# B&R Automation Studio project Pachore_Mayuresh_Project_3
Automation Studio 4.12.6.106; technology packages: Acp10Arnc0 5.24.1, mapp 5.24.1, mappView 5.24.4

## Configuration Config1

CPU 4PP065.0351-P74, AutomationRuntime B4.91, Build 4.1.2, Safety 1.10, Vc V4.73.2

### Task classes (Cpu.sw)
```
Cyclic#1:
  Main_Contr <- Main_Control.prg
Cyclic#2:
  Input_Brid <- Input_Bridge.prg
  Output_Bri <- Output_Bridge.prg
  Pallet <- Pallet.prg
  Crane <- Crane.prg
  Feeder <- Feeder.prg
  ComTCP_P <- Libraries.ComTCP.ComTCP_P.prg
Cyclic#4:
  Signal_Man <- Signal_Mangement.prg
Binaries: udbdef, mvLoader, FWRules, TCData, TCLang, sysconf, Role, User, iomap, ashwd, asfw, arconfig, ashwac, TC
Libraries: operator, astime, standard, AsArLog, AsBrStr, AsTCP, ComTCP_L, Signal_Mng, Gen_Axis, Gen_Device, fileio, asieccon, arssl, sys_lib, runtime, Blink, S_filter
```

### Hardware
```
4PP065_0351_P74 : 4PP065.0351-P74 v1.1.0.0
  Connector IF4:
    DNAConfiguration = manual
  Connector IF5:
    ActivateDevice = 1
  ConfigurationID = Pachore_Mayuresh_Project_3_Config1
  UserPartitionSize = 0
  Simulation = 1
  FileDevice1
  FileDeviceName1 = USER
  FileDevicePath1 = USER_PATH
  ActivateOpcUa = 1
  OpcUaInformationModels_PV_Version = 1
  KeyMappingFile = VC\4PP065_0351_P74.dis
```

### Acp10cfg.ncc - 4PP065_0351_P74/Motion/Acp10cfg.ncc
```
NcConfiguration (Version=5.24.1, NcSwId=Acp10)
  ACP10CF1_typ:
    cnt_nettrc_rec_drive = 150
    bufsize_trace_upload = 1200
    tc_nc_man_task = Cyclic #1
    glob_pv_as_ncobject = Yes
    ncsys_dl_broadcast = Yes
    ncsys_dl_acp_reset = Yes
    safemc_log_err_to_ax = Yes
    network_init:
      ncsw_init_execute = Yes
      automatic_execute = No
      node_nr_warning = Yes
      net_err_before_ncact = Yes
    nettrc:
      enter_parsecrec = Yes
      enter_ncaction = Yes
      save_ring_startidx = No
    cam_prof_download:
      cam_dat_dl_parallel = No
      tc_cam_dl_parallel = Task class for NC Manager task
```

### Acp10map.ncm - 4PP065_0351_P74/Motion/Acp10map.ncm
```
NcMapping (NcSwId=Acp10)
```

## Logical view

Binary libraries used (declarations not repeated): operator, runtime, astime, AsIecCon, Acp10man, Acp10par, NcGlobal, AsTCP, standard, AsArLog, AsBrStr, sys_lib

### MNG_Package.typ
```iecst
(*                                                                            *)
(* File generated by the B&R AS 4 control config generator                    *)
(*                                                                            *)
(*     Provider: machineering                                                 *)
(*  Application: industrialPhysics_2.4.master                                 *)
(* Architecture: Windows 64 Bit                                               *)
(*      Version: 2.4.10491.master                                             *)
(*        Build: 164f85bec                                                    *)
(*         Date: 2020-05-19, Time: 12:11:21                                   *)
(*                                                                            *)

TYPE
ComTCP_INPUTS_32BIT : STRUCT

		NumSignals	: INT := 15;

        laser_sensor_IR : BOOL := 0;
        (* BOOL laser_sensor_IR *)
        laser_sensor2_IR : BOOL := 0;
        (* BOOL laser_sensor2_IR *)
        carriage_2_AXIS : REAL := 0.0;
        (* REAL carriage_2_AXIS *)
        carriage_2_RCHD : BOOL := 0;
        (* BOOL carriage_2_RCHD *)
        turnpusher_LBK : BOOL := 0;
        (* BOOL turnpusher_LBK *)
        turnpusher_LFR : BOOL := 0;
        (* BOOL turnpusher_LFR *)
        gantry_crane_AXIS : REAL := 0.0;
        (* REAL gantry_crane_AXIS *)
        box_crane_AXIS : REAL := 0.0;
        (* REAL box_crane_AXIS *)
        vaccum_box_crane_VACUUM : BOOL := 0;
        (* BOOL vaccum_box_crane_VACUUM *)
        pallet_light_barrier_1_IR : BOOL := 0;
        (* BOOL pallet_light_barrier_1_IR *)
        pallet_light_barrier_2_IR : BOOL := 0;
        (* BOOL pallet_light_barrier_2_IR *)
        pusher_LBK : BOOL := 0;
        (* BOOL pusher_LBK *)
        pusher_LFR : BOOL := 0;
        (* BOOL pusher_LFR *)
        pallet_lifter_AXIS : REAL := 0.0;
        (* REAL pallet_lifter_AXIS *)
        pallet_fork_left_FB : BOOL := 0;
        (* BOOL pallet_fork_left_FB *)

	END_STRUCT;

ComTCP_OUTPUTS_32BIT : STRUCT

		NumSignals	: INT := 18;

        cartboard_TRIG : BOOL := 0;
        (* BOOL cartboard_TRIG *)
        conveyor_if_FWD : BOOL := 0;
        (* BOOL conveyor_if_FWD *)
        conveyer_turn1_FWD : BOOL := 0;
        (* BOOL conveyer_turn1_FWD *)
        conveyer_end_FWD : BOOL := 0;
        (* BOOL conveyer_end_FWD *)
        carriage_2_TGT_POS : REAL := 0.0;
        (* REAL carriage_2_TGT_POS *)
        turnpusher_FWD : BOOL := 0;
        (* BOOL turnpusher_FWD *)
        turnpusher_BWD : BOOL := 0;
        (* BOOL turnpusher_BWD *)
        gantry_crane_TGT_POS : REAL := 0.0;
        (* REAL gantry_crane_TGT_POS *)
        box_crane_TGT_POS : REAL := 0.0;
        (* REAL box_crane_TGT_POS *)
        slide_rail_right_EN : BOOL := 0;
        (* BOOL slide_rail_right_EN *)
        vaccum_box_crane_GRIP : BOOL := 0;
        (* BOOL vaccum_box_crane_GRIP *)
        pusher_z_EN : BOOL := 0;
        (* BOOL pusher_z_EN *)
        pusher_x_EN : BOOL := 0;
        (* BOOL pusher_x_EN *)
        pallet_conveyor_2_ACT_VEL : REAL := 0.0;
        (* REAL pallet_conveyor_2_ACT_VEL *)
        pusher_FW : BOOL := 0;
        (* BOOL pusher_FW *)
        pallet_lifter_TGT_POS : REAL := 0.0;
        (* REAL pallet_lifter_TGT_POS *)
        pallet_fork_left_EN : BOOL := 0;
        (* BOOL pallet_fork_left_EN *)
        pallet_conveyor_1_FWD : BOOL := 0;
        (* BOOL pallet_conveyor_1_FWD *)

	END_STRUCT;

END_TYPE
```

### MNG_Package.var
```iecst
(*                                                                            *)
(* File generated by the B&R AS 4 control config generator                    *)
(*                                                                            *)
(*     Provider: machineering                                                 *)
(*  Application: industrialPhysics_2.4.master                                 *)
(* Architecture: Windows 64 Bit                                               *)
(*      Version: 2.4.10491.master                                             *)
(*        Build: 164f85bec                                                    *)
(*         Date: 2020-05-19, Time: 12:11:21                                   *)
(*                                                                            *)

                VAR
                ComTCP_SimInputs : ComTCP_INPUTS_32BIT := (0);
    ComTCP_SimOutputs : ComTCP_OUTPUTS_32BIT := (0);

    ComTCP_SimServerAddress : STRING[15] := '127.0.0.1';
    ComTCP_SimServerPort : UINT := 5000;
    ComTCP_SimSendCycleTime : TIME := T#5ms;
    ComTCP_SimActive : BOOL := FALSE;

                END_VAR
```

### Global.var - Global variables
```iecst
(*Simulation Variables*)
(*Input Variables*)
VAR
	I_IR_Sensor_1 : BOOL := FALSE; (*laser_sensor_IR*)
	I_IR_Sensor_2 : BOOL := FALSE; (*laser_sensor2_IR*)
	I_Carriage_Push_Act_Pos : REAL := 1; (*carriage_2_AXIS*)
	I_Carriage_Push_Tar_Rec : BOOL := TRUE; (*carriage_2_RCHD*)
	I_Pusher_1_B : BOOL := FALSE; (*pusher_LBK*)
	I_Pusher_1_F : BOOL := TRUE; (*pusher_LFR*)
	I_Turn_Push_B : BOOL := FALSE; (*turnpusher_LBK*)
	I_Turn_Push_F : BOOL := TRUE; (*turnpusher_LFR*)
	I_Gantry_Crane_Act_Pos : REAL := 0; (*gantry_crane_AXIS*)
	I_Box_Crane_Act_Pos : REAL := 0; (*box_crane_AXIS*)
	I_Vacuum_retention_act : BOOL := FALSE; (*vacuum_box_crane_VACUUM*)
	I_Pallet_lift_Act_Pos : REAL := 0; (*pallet_lifter_AXIS*)
	I_Pallet_holder_State : BOOL := FALSE; (*pallet_fork_left_FB*)
	I_IR_Sensor_3 : BOOL := FALSE; (*pallet_light_barrier_1_IR*)
	I_IR_Sensor_4 : BOOL := FALSE; (*pallet_light_barrier_2_IR*)
END_VAR
(*Output Variables*)
VAR
	O_Conveyor_1 : BOOL := FALSE; (*Conveyor_if control*)
	O_Pusher_1 : BOOL := FALSE; (*pusher control*)
	O_Conveyor_2 : BOOL := FALSE; (*conveyor_turn1 control*)
	O_Conveyor_3 : BOOL := FALSE; (*conveyor_end control*)
	O_Turn_Pusher_ON : BOOL := FALSE; (*turnpusher Forward*)
	O_Turn_Pusher_OFF : BOOL := FALSE; (*turnpusher Backward*)
	O_Carriage_Tar_Pos : REAL := 0; (*carriage_2 control*)
	O_Gantry_Crane_Tar_Pos : REAL := 0; (*gantry_crane control*)
	O_Box_Crane_Tar_Pos : REAL := 0; (*box_crane control*)
	O_Cartboard_Trig : BOOL := FALSE; (*cartboard control*)
	O_Vacuum_Grip_act : BOOL := FALSE; (*vacuum_box_crane control*)
	O_Box_Holder : BOOL := FALSE; (*slide_rail_right control*)
	O_Pusher_z : BOOL := FALSE; (*pusher_z control*)
	O_Pusher_x : BOOL := FALSE; (*pusher_x control*)
	O_Pallet_lift_Tar_Pos : REAL := 0; (*pallet_lifter control*)
	O_Pallet_Holder : BOOL := FALSE; (*pallet_fork control*)
	O_Conveyor_4 : BOOL := FALSE; (*pallet_conveyor_1 control*)
	O_Conveyor_5_vel : REAL := 0; (*pallet_conveyor_2 control*)
END_VAR
(*HMI Variables*)
VAR
	Service_Mode_HMI : BOOL;
	Conveyor_1_Jog_HMI : BOOL;
	Pusher_1_Jog_HMI : BOOL;
	Conveyor_2_Jog_HMI : BOOL;
	Conveyor_3_Jog_HMI : BOOL;
	Conveyor_1_HMI : BOOL;
	Pusher_1_HMI : BOOL;
	Conveyor_2_HMI : BOOL;
	Conveyor_3_HMI : BOOL;
	Turn_Pusher_ON_HMI : BOOL;
	Turn_Pusher_OFF_HMI : BOOL;
	Carriage_Push_Origin_HMI : BOOL;
	Carriage_Push_Target_HMI : BOOL;
	Carriage_Target_Pos_HMI : REAL;
	Carriage_Tar_Pos_Dis_HMI : REAL;
	IR1_HMI : BOOL;
	IR2_HMI : BOOL;
	Turn_Pusher_F_HMI : BOOL;
	Turn_Pusher_B_HMI : BOOL;
	Pusher_1_F_HMI : BOOL;
	Pusher_1_B_HMI : BOOL;
	Carriage_Push_TarRech_HMI : BOOL;
	Carriage_Push_ActPos_Dis_HMI : REAL;
	vaccume_box_crane_grip_HMI : BOOL;
	Cartboard_Trig_HMI : BOOL;
	Slide_rail_right_EN_HMI : BOOL;
	pusher_z_EN_HMI : BOOL;
	pusher_x_EN_HMI : BOOL;
	gantry_crane_Origin_pos_HMI : BOOL;
	gantry_crane_TGT_pos_HMI : BOOL;
	gantry_crane_TGT_HMI : REAL;
	gantry_crane_TGT_dis_HMI : REAL;
	box_crane_TGT_pos_HMI : BOOL;
	box_crane_Origin_pos_HMI : BOOL;
	box_crane_TGT_HMI : REAL;
	box_crane_TGT_dis_HMI : REAL;
	vaccume_box_crane_state_HMI : BOOL;
	gantry_crane_Act_Pos_HMI : REAL;
	box_crane_Act_Pos_HMI : REAL;
	Pallet_fork_HMI : BOOL;
	Conveyor_4_Jog_HMI : BOOL;
	Conveyor_4_HMI : BOOL;
	Conveyor_5_S1_HMI : BOOL;
	Conveyor_5_S2_HMI : BOOL;
	Pallet_Lifter_Origin_pos_HMI : BOOL;
	Pallet_Lifter_TGT_pos_HMI : BOOL;
	Pallet_Lifter_TGT_HMI : REAL;
	Pallet_Lifter_TGT_dis_HMI : REAL;
	Pallet_Holder_State_HMI : BOOL;
	IR_3_HMI : BOOL;
	IR_4_HMI : BOOL;
	On_Phase_Stop_HMI : BOOL;
	Emergency_Stop_HMI : BOOL;
	Priority_4_HMI : STRING[80];
	Priority_3_HMI : STRING[80];
	Priority_2_HMI : STRING[80];
	Priority_1_HMI : STRING[80];
	Pallet_Lifter_Act_Pos_HMI : REAL;
END_VAR
(*Signal_Mng_Faults*)
VAR
	Operation_Type : INT := 0;
	Out_Of_Material : BOOL;
	Crane_Cartboard_Counter : INT := 3;
	Pallet_Counter : INT := 5;
	e_Turn_Pusher_Fault : BOOL := FALSE;
	e_Feeder_Pusher_Fault : BOOL := FALSE;
	e_Crane_Pusher_x_Fault : BOOL := FALSE;
	e_Crane_Pusher_z_Fault : BOOL := FALSE;
	e_Vacuum_Fault : BOOL := FALSE;
	e_Pallet_Fork_Fault : BOOL := FALSE;
	e_Carriage_Fault : BOOL := FALSE;
	e_Gantry_Crane_Fault : BOOL := FALSE;
	e_Box_Crane_Fault : BOOL := FALSE;
	e_Pallet_Lifter_Fault : BOOL := FALSE;
	e_Conveyor_1_Fault : BOOL := FALSE;
	e_Conveyor_2_Fault : BOOL := FALSE;
	e_Conveyor_3_Fault : BOOL := FALSE;
	e_Cartboard_Fault : BOOL := FALSE;
	e_Box_Holder_Fault : BOOL := FALSE;
	e_Conveyor_4_Fault : BOOL := FALSE;
	e_Conveyor_5_Fault : BOOL := FALSE;
	Fault : ARRAY[0..23] OF STRING[80] := ['',2('Feeder Fault Technician Required'),3('Crane Fault Technician Required'),'Pallet Fault Technician Required','Pallet Refill Required','Feeder Fault Technician Required',2('Crane Fault Technician Required'),'Pallet Fault Technician Required','Prepare Pallets to Refill','On Phase Stop Requested','Emergency Stop Requested','Prepare Cartboards to Refill','Cartboard Refill Required',3('Feeder Fault Technician Required'),2('Crane Fault Technician Required'),2('Pallet Fault Technician Required')];
END_VAR
(*Main*)
VAR
	Service_Mode : BOOL;
	En_Machine : BOOL := FALSE;
	Start_Machine : BOOL := FALSE;
	Emergency_Stop : BOOL;
	Immediate_Stop : BOOL;
	On_Phase_Stop : BOOL;
	Hold_Boxes : BOOL;
	P_Exit_Done : BOOL;
	Boxes_On_The_P : BOOL;
	Boxes_On_The_C : BOOL; (*Feeder*)
	Load_Boxes_On_The_C : BOOL; (*Feeder*)
	Load_Boxes_On_The_P : BOOL;
	Second_Layer : BOOL; (*Feeder*)
	M_Current_State : STRING[80];
	P_Exit_En : BOOL;
END_VAR
(*Communication between Feeder and Main*)
VAR
	Start_Feeder : BOOL := FALSE;
	F_Emergency_Stop : BOOL := FALSE;
	F_Reset_Config : BOOL := FALSE;
	F_Immediate_Stop : BOOL := FALSE;
	F_On_Phase_Stop : BOOL := FALSE;
	F_Restart : BOOL := FALSE;
	F_Ready : BOOL := FALSE;
END_VAR
(*Communication between Crane and Main*)
VAR
	Start_Crane : BOOL := FALSE;
	C_Reset_Config : BOOL := FALSE;
	C_Emergency_Stop : BOOL := FALSE;
	C_Immediate_Stop : BOOL := FALSE;
	C_On_Phase_Stop : BOOL := FALSE;
	C_Restart : BOOL := FALSE;
	C_Ready : BOOL := FALSE;
END_VAR
(*Communication between Pallet and Main*)
VAR
	Start_Pallet : BOOL := FALSE;
	P_Emergency_Stop : BOOL := FALSE;
	P_Reset_Config : BOOL := FALSE;
	P_Immediate_Stop : BOOL := FALSE;
	P_On_Phase_Stop : BOOL := FALSE;
	P_Restart : BOOL := FALSE;
	P_Ready : BOOL := FALSE;
END_VAR
(*Feeder Variables*)
VAR
	Conveyor_3_Fault_HMI : BOOL;
	Conveyor_2_Fault_HMI : BOOL;
	Conveyor_1_Fault_HMI : BOOL;
	Turn_Pusher_Fault_HMI : BOOL;
	Carriage_Fault_HMI : BOOL;
	Pusher_1_Fault_HMI : BOOL;
	Box_Counter : INT := 0;
	C_Layer_Counter : BOOL := FALSE;
	End_Layer : BOOL;
	F_Current_State : STRING[80];
END_VAR
(*Crane Variables*)
VAR
	Gantry_Crane_Fault_HMI : BOOL;
	Box_Crane_Fault_HMI : BOOL;
	Cartboard_Fault_HMI : BOOL;
	Vacuum_Fault_HMI : BOOL;
	Box_Holder_Fault_HMI : BOOL;
	Crane_Pusher_X_Fault_HMI : BOOL;
	Crane_Pusher_Z_Fault_HMI : BOOL;
	C_Current_State : STRING[80];
END_VAR
(*Pallet Variables*)
VAR
	Pallet_Lifter_Fault_HMI : BOOL;
	Pallet_Fork_Fault_HMI : BOOL;
	Pallet_Conv_1_Fault_HMI : BOOL;
	Pallet_Conv_2_Fault_HMI : BOOL;
	P_Current_State : STRING[80];
END_VAR
(*LED Blinker*)
VAR
	Reset_Unlocked : BOOL;
	Aux_Reset_Unlocked : BOOL;
	Aux_Unlocked : Blink;
	R_Unlocked : Blink;
	Warning_Detected : Blink;
	Alarm_Detected : Blink;
END_VAR
```

### Package Logical/Libraries - Global libraries

### Library Logical/Libraries/ComTCP/ComTCP_L (ANSIC)
Depends on: AsTCP, operator, runtime, astime, standard, AsArLog, AsBrStr, Convert

#### MNG_ComHdlr.hpp
```cpp
#ifndef _MNGCOMHDLR_HPP_
#define _MNGCOMHDLR_HPP_

#define TRUE  1
#define FALSE 0

#include "MNG_InternalTyp.hpp"

#include <bur/plc.h>
#include <bur/plctypes.h>
#include <AsTCP.h>
#include <standard.h>
#include <astime.h>
#include <runtime.h>
#include <AsBrStr.h>

typedef struct{
	TcpOpen_typ tcpOpen;
	TcpIoctl_typ tcpIoctl;
	tcpLINGER_typ tcpLINGER;
	TcpSend_typ tcpSend;
	TcpClose_typ tcpClose;
	TcpRecv_typ tcpRecv;
	TcpClient_typ tcpClient;
} asTcpFcn_t;

typedef enum {
	MNG_wSock,
	MNG_skippedMessage
} MNG_errorCases;

typedef enum {
	MNG_Init,
	MNG_Socket,
	MNG_Open,
	MNG_SetIo,
	MNG_Linger,
	MNG_Connecting,
	MNG_Exchange,
	MNG_Closing,
        MNG_Reset
} MNG_internalState_t;

	extern unsigned long int MNG_CpyOutToMsg(MNG_RawDatagram * pToServer, unsigned long int counter, ComTCP_OUTPUTS_32BIT_FWRD *pSimOutputs);
	extern unsigned long int MNG_CpyMsgToInp(MNG_RawDatagram * pFromServer, ComTCP_INPUTS_32BIT_FWRD *pSimInputs);

class MNG_ComHdlr
{
	public:

	MNG_ComHdlr(char *srvIpAdr, unsigned int srvPort, TIME sendCycleTime);
	~MNG_ComHdlr();

        int RunCommunication(void*, void*, BOOL*);

	private:

	char* _srvIpAdr;
	unsigned int _srvPort;
	TIME _sendCycleTime;

	unsigned int _error;

	MNG_internalState_t _internalState;
	TON_typ _connectionTon;
	TIME _connectionTime;

	bool _connect;
	bool _sendDone;

	signed int _recvOffset;

	signed long int _potMsgLen;
	signed long int _totalRecvLen;

	unsigned long int _one;
	unsigned long int _counter;
	unsigned long int _recvLen;
	unsigned long int _recvBuffer[10000];
	TON_typ _sendTon;
	MNG_RawDatagram _recvMessage;
	MNG_RawDatagram _sendMessage;

	static const signed long int SIXTEEN = 16;
	static const unsigned int PORT = 0;
	static const unsigned long int MNG_MAXPAYLOAD = 1400;

	void init_TcpOpen();
	void init_TcpSocket();
	void init_TcpIoctl();
	void init_TcpLinger();
	void init_TcpClient();
	void init_TcpRecv();
	void init_TcpSend(ComTCP_OUTPUTS_32BIT_FWRD* pSimOut);

	void InitParams();

	void SetSendDone(bool toogle);
	void SetStateValue(MNG_internalState_t stateVal);

};
#endif
```

#### MNG_Global.hpp
```cpp
#ifndef  _MNGGLOBAL_HPP_
#define _MNGGLOBAL_HPP_

#include <mng_globalTYP.h>

    typedef struct {

		signed short NumSignals;

        /* BOOL laser_sensor_IR */
        BOOL laser_sensor_IR;
        /* BOOL laser_sensor2_IR */
        BOOL laser_sensor2_IR;
        /* REAL carriage_2_AXIS */
        REAL carriage_2_AXIS;
        /* BOOL carriage_2_RCHD */
        BOOL carriage_2_RCHD;
        /* BOOL turnpusher_LBK */
        BOOL turnpusher_LBK;
        /* BOOL turnpusher_LFR */
        BOOL turnpusher_LFR;
        /* REAL gantry_crane_AXIS */
        REAL gantry_crane_AXIS;
        /* REAL box_crane_AXIS */
        REAL box_crane_AXIS;
        /* BOOL vaccum_box_crane_VACUUM */
        BOOL vaccum_box_crane_VACUUM;
        /* BOOL pallet_light_barrier_1_IR */
        BOOL pallet_light_barrier_1_IR;
        /* BOOL pallet_light_barrier_2_IR */
        BOOL pallet_light_barrier_2_IR;
        /* BOOL pusher_LBK */
        BOOL pusher_LBK;
        /* BOOL pusher_LFR */
        BOOL pusher_LFR;
        /* REAL pallet_lifter_AXIS */
        REAL pallet_lifter_AXIS;
        /* BOOL pallet_fork_left_FB */
        BOOL pallet_fork_left_FB;

        } ComTCP_INPUTS_32BIT_FWRD;

    typedef struct {

		signed short NumSignals;

        /* BOOL cartboard_TRIG */
        BOOL cartboard_TRIG;
        /* BOOL conveyor_if_FWD */
        BOOL conveyor_if_FWD;
        /* BOOL conveyer_turn1_FWD */
        BOOL conveyer_turn1_FWD;
        /* BOOL conveyer_end_FWD */
        BOOL conveyer_end_FWD;
        /* REAL carriage_2_TGT_POS */
        REAL carriage_2_TGT_POS;
        /* BOOL turnpusher_FWD */
        BOOL turnpusher_FWD;
        /* BOOL turnpusher_BWD */
        BOOL turnpusher_BWD;
        /* REAL gantry_crane_TGT_POS */
        REAL gantry_crane_TGT_POS;
        /* REAL box_crane_TGT_POS */
        REAL box_crane_TGT_POS;
        /* BOOL slide_rail_right_EN */
        BOOL slide_rail_right_EN;
        /* BOOL vaccum_box_crane_GRIP */
        BOOL vaccum_box_crane_GRIP;
        /* BOOL pusher_z_EN */
        BOOL pusher_z_EN;
        /* BOOL pusher_x_EN */
        BOOL pusher_x_EN;
        /* REAL pallet_conveyor_2_ACT_VEL */
        REAL pallet_conveyor_2_ACT_VEL;
        /* BOOL pusher_FW */
        BOOL pusher_FW;
        /* REAL pallet_lifter_TGT_POS */
        REAL pallet_lifter_TGT_POS;
        /* BOOL pallet_fork_left_EN */
        BOOL pallet_fork_left_EN;
        /* BOOL pallet_conveyor_1_FWD */
        BOOL pallet_conveyor_1_FWD;

        } ComTCP_OUTPUTS_32BIT_FWRD;

#endif
```

#### MNG_CpyOutToMsg.cpp
```cpp
#include "MNG_InternalTyp.hpp"

unsigned long int MNG_CpyOutToMsg(MNG_RawDatagram * pToServer, unsigned long int counter, ComTCP_OUTPUTS_32BIT_FWRD *pSimOutputs ) {

        unsigned long int DWordBuffer;

        pSimOutputs->NumSignals = 18;
        (pToServer->Header).ByteCount    = H_TO_NUDINT(76);
        (pToServer->Header).DatagramType = H_TO_NUDINT(MNG_Raw32BitImage);
        (pToServer->Header).SentTime = H_TO_NUDINT(0);  // Todo
        (pToServer->Header).Counter = H_TO_NUDINT(counter);
        pToServer->Payload[0] = H_TO_NUDINT(pSimOutputs->NumSignals);

    /* cartboard_TRIG : BOOL */
    if(pSimOutputs->cartboard_TRIG == 1) {
        pToServer->Payload[1] = 0xFFFFFFFF;   /*BOOL */
    } else {
        pToServer->Payload[1] = 0;
    }

    /* conveyor_if_FWD : BOOL */
    if(pSimOutputs->conveyor_if_FWD == 1) {
        pToServer->Payload[2] = 0xFFFFFFFF;   /*BOOL */
    } else {
        pToServer->Payload[2] = 0;
    }

    /* conveyer_turn1_FWD : BOOL */
    if(pSimOutputs->conveyer_turn1_FWD == 1) {
        pToServer->Payload[3] = 0xFFFFFFFF;   /*BOOL */
    } else {
        pToServer->Payload[3] = 0;
    }

    /* conveyer_end_FWD : BOOL */
    if(pSimOutputs->conveyer_end_FWD == 1) {
        pToServer->Payload[4] = 0xFFFFFFFF;   /*BOOL */
    } else {
        pToServer->Payload[4] = 0;
    }

    /* carriage_2_TGT_POS : FLOAT32 */
    brsmemcpy((unsigned long int)&(DWordBuffer), (unsigned long int)&(pSimOutputs->carriage_2_TGT_POS), 4);
    pToServer->Payload[5] = H_TO_NUDINT(DWordBuffer);

    /* turnpusher_FWD : BOOL */
    if(pSimOutputs->turnpusher_FWD == 1) {
        pToServer->Payload[6] = 0xFFFFFFFF;   /*BOOL */
    } else {
        pToServer->Payload[6] = 0;
    }

    /* turnpusher_BWD : BOOL */
    if(pSimOutputs->turnpusher_BWD == 1) {
        pToServer->Payload[7] = 0xFFFFFFFF;   /*BOOL */
    } else {
        pToServer->Payload[7] = 0;
    }

    /* gantry_crane_TGT_POS : FLOAT32 */
    brsmemcpy((unsigned long int)&(DWordBuffer), (unsigned long int)&(pSimOutputs->gantry_crane_TGT_POS), 4);
    pToServer->Payload[8] = H_TO_NUDINT(DWordBuffer);

    /* box_crane_TGT_POS : FLOAT32 */
    brsmemcpy((unsigned long int)&(DWordBuffer), (unsigned long int)&(pSimOutputs->box_crane_TGT_POS), 4);
    pToServer->Payload[9] = H_TO_NUDINT(DWordBuffer);

    /* slide_rail_right_EN : BOOL */
    if(pSimOutputs->slide_rail_right_EN == 1) {
        pToServer->Payload[10] = 0xFFFFFFFF;   /*BOOL */
    } else {
        pToServer->Payload[10] = 0;
    }

    /* vaccum_box_crane_GRIP : BOOL */
    if(pSimOutputs->vaccum_box_crane_GRIP == 1) {
        pToServer->Payload[11] = 0xFFFFFFFF;   /*BOOL */
    } else {
        pToServer->Payload[11] = 0;
    }

    /* pusher_z_EN : BOOL */
    if(pSimOutputs->pusher_z_EN == 1) {
        pToServer->Payload[12] = 0xFFFFFFFF;   /*BOOL */
    } else {
        pToServer->Payload[12] = 0;
    }

    /* pusher_x_EN : BOOL */
    if(pSimOutputs->pusher_x_EN == 1) {
        pToServer->Payload[13] = 0xFFFFFFFF;   /*BOOL */
    } else {
        pToServer->Payload[13] = 0;
    }

    /* pallet_conveyor_2_ACT_VEL : FLOAT32 */
    brsmemcpy((unsigned long int)&(DWordBuffer), (unsigned long int)&(pSimOutputs->pallet_conveyor_2_ACT_VEL), 4);
    pToServer->Payload[14] = H_TO_NUDINT(DWordBuffer);

    /* pusher_FW : BOOL */
    if(pSimOutputs->pusher_FW == 1) {
        pToServer->Payload[15] = 0xFFFFFFFF;   /*BOOL */
    } else {
        pToServer->Payload[15] = 0;
    }

    /* pallet_lifter_TGT_POS : FLOAT32 */
    brsmemcpy((unsigned long int)&(DWordBuffer), (unsigned long int)&(pSimOutputs->pallet_lifter_TGT_POS), 4);
    pToServer->Payload[16] = H_TO_NUDINT(DWordBuffer);

    /* pallet_fork_left_EN : BOOL */
    if(pSimOutputs->pallet_fork_left_EN == 1) {
        pToServer->Payload[17] = 0xFFFFFFFF;   /*BOOL */
    } else {
        pToServer->Payload[17] = 0;
    }

    /* pallet_conveyor_1_FWD : BOOL */
    if(pSimOutputs->pallet_conveyor_1_FWD == 1) {
        pToServer->Payload[18] = 0xFFFFFFFF;   /*BOOL */
    } else {
        pToServer->Payload[18] = 0;
    }

	return 0;
}
```

#### MNG_CpyMsgToInp.cpp
```cpp
#include "MNG_InternalTyp.hpp"

unsigned long int MNG_CpyMsgToInp(MNG_RawDatagram * pFromServer, ComTCP_INPUTS_32BIT_FWRD *pSimInputs) {

    MNG_DatagramType datagramType;
	unsigned long int DWordBuffer;
        unsigned long int byteCount;
	unsigned long int numSignalsInMessage;

	byteCount = N_TO_HUDINT((pFromServer->Header).ByteCount);
	datagramType = static_cast<MNG_DatagramType>(N_TO_HUDINT((pFromServer->Header).DatagramType));
	if (datagramType != MNG_Raw32BitImage) {
		return 0;
	}

    pSimInputs->NumSignals = 15;

    numSignalsInMessage = N_TO_HUDINT(pFromServer->Payload[0]);
        if ((static_cast<long int>(numSignalsInMessage) != pSimInputs->NumSignals) ||
	(byteCount != 4 + numSignalsInMessage * 4)) {
		return 0;
	}

    /* BOOL laser_sensor_IR */
    pSimInputs->laser_sensor_IR = (pFromServer->Payload[1] != 0);

    /* BOOL laser_sensor2_IR */
    pSimInputs->laser_sensor2_IR = (pFromServer->Payload[2] != 0);

    /* FLOAT32 carriage_2_AXIS */
    DWordBuffer = N_TO_HUDINT(pFromServer->Payload[3]);
    brsmemcpy((unsigned long int)&(pSimInputs->carriage_2_AXIS), (unsigned long int)&(DWordBuffer), 4);

    /* BOOL carriage_2_RCHD */
    pSimInputs->carriage_2_RCHD = (pFromServer->Payload[4] != 0);

    /* BOOL turnpusher_LBK */
    pSimInputs->turnpusher_LBK = (pFromServer->Payload[5] != 0);

    /* BOOL turnpusher_LFR */
    pSimInputs->turnpusher_LFR = (pFromServer->Payload[6] != 0);

    /* FLOAT32 gantry_crane_AXIS */
    DWordBuffer = N_TO_HUDINT(pFromServer->Payload[7]);
    brsmemcpy((unsigned long int)&(pSimInputs->gantry_crane_AXIS), (unsigned long int)&(DWordBuffer), 4);

    /* FLOAT32 box_crane_AXIS */
    DWordBuffer = N_TO_HUDINT(pFromServer->Payload[8]);
    brsmemcpy((unsigned long int)&(pSimInputs->box_crane_AXIS), (unsigned long int)&(DWordBuffer), 4);

    /* BOOL vaccum_box_crane_VACUUM */
    pSimInputs->vaccum_box_crane_VACUUM = (pFromServer->Payload[9] != 0);

    /* BOOL pallet_light_barrier_1_IR */
    pSimInputs->pallet_light_barrier_1_IR = (pFromServer->Payload[10] != 0);

    /* BOOL pallet_light_barrier_2_IR */
    pSimInputs->pallet_light_barrier_2_IR = (pFromServer->Payload[11] != 0);

    /* BOOL pusher_LBK */
    pSimInputs->pusher_LBK = (pFromServer->Payload[12] != 0);

    /* BOOL pusher_LFR */
    pSimInputs->pusher_LFR = (pFromServer->Payload[13] != 0);

    /* FLOAT32 pallet_lifter_AXIS */
    DWordBuffer = N_TO_HUDINT(pFromServer->Payload[14]);
    brsmemcpy((unsigned long int)&(pSimInputs->pallet_lifter_AXIS), (unsigned long int)&(DWordBuffer), 4);

    /* BOOL pallet_fork_left_FB */
    pSimInputs->pallet_fork_left_FB = (pFromServer->Payload[15] != 0);

return N_TO_HUDINT((pFromServer->Header).Counter); // return counter
}
```

### Program Logical/Libraries/ComTCP/ComTCP_P

#### Main.cpp
```cpp
#include <bur/plctypes.h>

#ifdef _DEFAULT_INCLUDES
        #include <AsDefault.h>
#endif

#include "../ComTCP_L/MNG_Global.hpp"
#include "../ComTCP_L/MNG_InternalTyp.hpp"
#include "../ComTCP_L/MNG_ComHdlr.hpp"

unsigned long bur_heap_size = 0xFFFF;

MNG_ComHdlr *pMNG_ComHdlr;

void _INIT ProgramInit(void)
{
    pMNG_ComHdlr = new MNG_ComHdlr(ComTCP_SimServerAddress, ComTCP_SimServerPort, ComTCP_SimSendCycleTime);
}

void _CYCLIC ProgramCyclic(void)
{
    connectionState = pMNG_ComHdlr->RunCommunication((void*)&ComTCP_SimInputs,(void*)&ComTCP_SimOutputs, &ComTCP_SimActive);
}

void _EXIT ProgramExit(void)
{
    delete pMNG_ComHdlr;
}
```

### Library Logical/Libraries/S_filter (IEC)

#### S_filter.fun - Exported functions and function blocks
```iecst
FUNCTION_BLOCK S_filter
	VAR_INPUT
		Sensor_Raw : BOOL;
		Sensor_Data : REAL;
		threshold_F : REAL;
		threshold_B : INT;
		Is_Bool : BOOL;
	END_VAR
	VAR_OUTPUT
		Sensor_Filtered : BOOL;
		Sensor_Data_Filtered : REAL;
	END_VAR
	VAR
		last_State : BOOL := FALSE;
		counter : INT := 0;
		init : BOOL := FALSE;
	END_VAR
END_FUNCTION_BLOCK
```

#### S_filter.st
```iecst
(* For Sensor Data Filter *)
FUNCTION_BLOCK S_filter
	IF Is_Bool THEN
		// BOOLEAN MODE filtering
		IF Sensor_Raw = last_State THEN
			counter := counter + 1;
		ELSE
			counter := 0;
			last_State := Sensor_Raw;
		END_IF;

		IF counter >= threshold_B THEN
			Sensor_Filtered := Sensor_Raw;
			counter := 0; // reset after output change
		END_IF;

	ELSE
		// REAL MODE: Exponential smoothing
		IF NOT init THEN
			Sensor_Data_Filtered := Sensor_Data;
			init := TRUE;
		ELSE
			Sensor_Data_Filtered := threshold_F * Sensor_Data + (1.0 - threshold_F) * Sensor_Data_Filtered;
		END_IF;
	END_IF;

END_FUNCTION_BLOCK
```

### Library Logical/Libraries/Signal_Mng (IEC)

#### Constants.var - Exported constants
```iecst
VAR CONSTANT
	Init : INT := 0;
	Run : INT := 1;
	Start_Configuration : INT := 2;
	Configuration : INT := 3;
	Start_Generation : INT := 4;
	Generation : INT := 5;
	Alarm : DINT := 2#0000000000000001;
	Anomaly : DINT := 2#0000000000000010;
	Warning : DINT := 2#0000000000000011;
	Information : DINT := 2#0000000000000100;
	Aux_Reset : DINT := 2#0000001000000000;
	Unconditioned_Reset : DINT := 2#0100000000000000;
	Auto_Conditioned_Reset : DINT := 2#0010000000000000;
	Auto_Provisional_Reset : DINT := 2#0001000000000000;
	Auto_Priority_Reset : DINT := 2#0000100000000000;
	Auto_Reset : DINT := 2#0000010000000000;
	Signal_Type_Mask : DINT := 2#0000000000000111;
	Sign_None : DWORD := 16#0000;
	Sign_Emergency_Stop : DWORD := 16#0001;
	Sign_Immediate_Stop : DWORD := 16#0002;
	Sign_On_Phase_Stop : DWORD := 16#0004;
	Sign_Machine_Out_Of_Phase : DWORD := 16#0100;
	Sign_Machine_Inhibition : DWORD := 16#0200;
	Sign_Materials_Run_Out_Lamp : DWORD := 16#0400;
	Sign_Materials_Run_Out_Buzzer : DWORD := 16#0800;
	Sign_IO_Diagostic_Inhibition : DWORD := 16#8000;
END_VAR
```

#### Signal_Mng.fun - Exported functions and function blocks
```iecst
FUNCTION_BLOCK Signal_Mng
	VAR_INPUT
		Operation_Type : INT;
		Signal_Type : DINT := 0;
		Signal_Code : INT := 0;
		Signal_Output : DWORD := 0;
		Activation_Signal : BOOL := FALSE;
		Auto_Reset_Signal : BOOL := FALSE;
		Reset : BOOL;
		Key_Reset : BOOL;
	END_VAR
	VAR_OUTPUT
		Signal_Outputs : DWORD;
		Signal_Priority_Code : WORD;
		Reset_Enable : BOOL;
		Aux_Reset_Enable : BOOL;
		Signal_Type_Alarm : BOOL;
		Signal_Type_Anomaly : BOOL;
		Signal_Type_Warning : BOOL;
		Signal_Type_Information : BOOL;
		Number_of_Alarms : INT;
		Number_of_Anomalies : INT;
		Number_of_Warnings : INT;
		Number_of_Information : INT;
		Active_Signal_Codes : ARRAY[1..30] OF INT;
		Number_of_Active_Alarms : INT := 0;
		Number_of_Active_Anomalies : INT := 0;
		Number_of_Active_Warning : INT := 0;
		Number_of_Active_Information : INT := 0;
		Signal_Mng_Error : BOOL;
		First_Signal_Index : INT;
		First_Active_Signal_Index : INT;
		Second_Active_Signal_Index : INT;
		Third_Active_Signal_Index : INT;
		Fourth_Active_Signal_Index : INT;
	END_VAR
	VAR
		Reset_Signals_Enable : BOOL;
		Aux_Reset_Activation : BOOL;
		Reset_Activation : BOOL;
		Signal_Request : BOOL;
		Signal_Ack_Request : BOOL;
		Signals : ARRAY[1..23] OF BOOL;
		Last_Signal_Index : INT;
		Active_Signal_Request : BOOL;
		Active_Signal_Request_Ack : BOOL;
		Last_Active_Signal_Index : INT;
		Reset_Old : BOOL;
		Key_Reset_Old : BOOL;
		Index : INT;
		Base_Index : INT;
		Condition : BOOL := FALSE;
		i : INT;
		Last_Information_Index : INT;
		Last_Anomaly_Index : INT;
		Last_Warning_Index : INT;
		Aux_Reset_Required : BOOL;
		d : INT := 1;
		Active_Signal : ARRAY[0..4] OF INT;
	END_VAR
END_FUNCTION_BLOCK
```

#### Signal_Mng.st
```iecst
FUNCTION_BLOCK Signal_Mng

	CASE Operation_Type OF

		Start_Configuration:
			Number_of_Alarms 		:= 0;
			Number_of_Anomalies 	:= 0;
			Number_of_Warnings 		:= 0;
			Number_of_Information 	:= 0;

		Configuration:
			CASE (Signal_Type AND Signal_Type_Mask) OF
				Alarm:
					Number_of_Alarms 		:= Number_of_Alarms + 1;
				Anomaly:
					Number_of_Anomalies		:= Number_of_Anomalies + 1;
				Warning:
					Number_of_Warnings 		:= Number_of_Warnings + 1;
				Information:
					Number_of_Information 	:= Number_of_Information + 1;
			END_CASE

		Start_Generation:
			Aux_Reset_Enable 		:= FALSE;
			Reset_Enable 			:= FALSE;
			Signal_Outputs 			:= Sign_None;
			Reset_Activation 		:= Reset AND NOT Reset_Old;
			Reset_Old 				:= Reset;
			Aux_Reset_Activation 	:= Key_Reset AND NOT Key_Reset_Old;
			Key_Reset_Old 			:= Key_Reset;

		Generation:
			CASE (Signal_Type AND Signal_Type_Mask) OF
				Alarm:
					Index 		:= Number_of_Active_Alarms;
					Base_Index 	:= 0;
					Condition 	:= TRUE;

				Anomaly:
					Index 		:= Number_of_Active_Anomalies;
					Base_Index 	:= Number_of_Alarms;
					Condition 	:= TRUE;

				Warning:
					Index 		:= Number_of_Active_Warning;
					Base_Index 	:= Number_of_Alarms + Number_of_Anomalies;
					Condition 	:= FALSE;

				Information:
					Index 		:= Number_of_Active_Information;
					Base_Index 	:= Number_of_Alarms + Number_of_Anomalies + Number_of_Warnings;
					Condition 	:= FALSE;
			END_CASE

			IF Activation_Signal AND NOT Signals[Signal_Code] THEN
				Signals[Signal_Code] 					:= TRUE;
				Index 									:= Index + 1;
				Active_Signal_Codes[Base_Index + Index] := Signal_Code;

			END_IF

			Aux_Reset_Required := ((Signal_Type AND Aux_Reset) = Aux_Reset);

			IF (Condition AND Signals[Signal_Code] AND NOT Activation_Signal AND (Active_Signal_Codes[Base_Index + 1] = Signal_Code) AND Aux_Reset_Required) THEN
				Aux_Reset_Enable 						:= TRUE;
			END_IF

			IF (Condition AND Signals[Signal_Code] AND NOT Activation_Signal AND (Active_Signal_Codes[Base_Index + 1] = Signal_Code) AND NOT Aux_Reset_Required) THEN
				Reset_Enable							:= TRUE;
			END_IF

			IF ((Reset_Activation OR NOT Condition) AND Signals[Signal_Code] AND NOT Activation_Signal AND (Active_Signal_Codes[Base_Index + 1] = Signal_Code) AND NOT Aux_Reset_Required) THEN
				Signals[Signal_Code] 					:= FALSE;

				FOR i := 2 TO Index DO
					Active_Signal_Codes[Base_Index + i-1] 	:= Active_Signal_Codes[Base_Index + i];
				END_FOR

				Active_Signal_Codes[Base_Index + Index] 	:= 0;
				Index 										:= Index - 1;
				Reset_Activation 							:= FALSE;
			END_IF

			IF ((Aux_Reset_Activation OR NOT Condition) AND Signals[Signal_Code] AND NOT Activation_Signal AND (Active_Signal_Codes[Base_Index + 1] = Signal_Code) AND Aux_Reset_Required) THEN
				Signals[Signal_Code] := FALSE;

				FOR i := 2 TO Index DO
					Active_Signal_Codes[Base_Index + i-1] := Active_Signal_Codes[Base_Index + i];
				END_FOR;

				Active_Signal_Codes[Base_Index + Index] := 0;
				Index := Index - 1;
				Aux_Reset_Activation := FALSE;
			END_IF

			CASE (Signal_Type AND Signal_Type_Mask) OF
				Alarm:
					Number_of_Active_Alarms 		:= Index;
				Anomaly:
					Number_of_Active_Anomalies 		:= Index;
				Warning:
					Number_of_Active_Warning 		:= Index;
				Information:
					Number_of_Active_Information 	:= Index;
			END_CASE

			IF Signals[Signal_Code] THEN
				Signal_Outputs := Signal_Outputs OR Signal_Output;
			END_IF

		Run:
			FOR d := 1 TO 4 DO
				Active_Signal[d] := 0;
			END_FOR

			d := 1;
			FOR i := 1 TO 30 DO
				IF Active_Signal_Codes[i] > 0 THEN
					Active_Signal[d] := Active_Signal_Codes[i];
					d := d + 1;
				END_IF
				IF d > 4 THEN
					EXIT;
				END_IF
			END_FOR

			First_Active_Signal_Index 		:= Active_Signal[1];
			Second_Active_Signal_Index 		:= Active_Signal[2];
			Third_Active_Signal_Index 		:= Active_Signal[3];
			Fourth_Active_Signal_Index 		:= Active_Signal[4];

			Last_Information_Index := Number_of_Alarms + Number_of_Anomalies + Number_of_Warnings + Number_of_Active_Information;
			IF Number_of_Active_Information > 0 THEN
				Signal_Type_Information 	:= TRUE;
			ELSE
				Signal_Type_Information 	:= FALSE;
			END_IF

			Last_Anomaly_Index 				:= Number_of_Alarms + Number_of_Anomalies + Number_of_Active_Anomalies;
			IF Number_of_Active_Anomalies > 0 THEN
				Signal_Type_Anomaly 		:= TRUE;
			ELSE
				Signal_Type_Anomaly 		:= FALSE;
			END_IF

			Last_Warning_Index 				:= Number_of_Alarms + Number_of_Active_Warning;
			IF Number_of_Active_Warning > 0 THEN
				Signal_Type_Warning 		:= TRUE;
			ELSE
				Signal_Type_Warning 		:= FALSE;
			END_IF

			IF Number_of_Active_Alarms > 0 THEN
				Signal_Type_Alarm 			:= TRUE;
			ELSE
				Signal_Type_Alarm 			:= FALSE;
			END_IF

	END_CASE

END_FUNCTION_BLOCK
```

### Library Logical/Libraries/Gen_Axis (IEC)

#### Types.typ - Exported data types
```iecst
TYPE
	AxisStateType :
		(
		Axis_Check_Command,
		Axis_Wait_TGT_Position,
		Axis_Wait_TGT_Velocity,
		Axis_Fault_State
		);
END_TYPE
```

#### Constants.var - Exported constants
```iecst
VAR CONSTANT
	Axis_Idle : WORD := 0;
	Axis_Change_Velocity : WORD := 1;
	Axis_Change_Position : WORD := 2;
	Axis_Emergency_Stop_Request : WORD := 3;
END_VAR
```

#### Gen_Axis.fun - Exported functions and function blocks
```iecst
FUNCTION_BLOCK Gen_Axis
	VAR_INPUT
		Axis_Command : WORD := 95;
		Axis_Act_Position : REAL;
		Axis_Act_Velocity : REAL;
		New_Set_Point : REAL;
		Axis_Dev_Timer : INT;
		Axis_TGT_Sensor : BOOL;
		Axis_Reset : BOOL;
	END_VAR
	VAR_OUTPUT
		Axis_TGT_Velocity : REAL;
		Axis_TGT_Position : REAL;
		Axis_In_Pos : BOOL;
		Axis_In_Vel : BOOL;
		Axis_Dev_Fault : BOOL;
	END_VAR
	VAR
		Axis_State : AxisStateType := Axis_Check_Command;
		Axis_Timer : INT;
	END_VAR
END_FUNCTION_BLOCK
```

#### Gen_Axis.st
```iecst
FUNCTION_BLOCK Gen_Axis

	CASE Axis_State OF

		Axis_Check_Command:

			IF Axis_Command 	 = Axis_Idle THEN
				Axis_In_Pos 	:= FALSE;
				Axis_In_Vel 	:= FALSE;
				Axis_Timer 		:= Axis_Dev_Timer;
				Axis_Dev_Fault 	:= FALSE;
			END_IF

			IF Axis_Command 		 = Axis_Change_Position THEN
				Axis_TGT_Position 	:= New_Set_Point;
				Axis_State 			:= Axis_Wait_TGT_Position;
			END_IF

			IF Axis_Command 		 = Axis_Change_Velocity THEN
				Axis_TGT_Velocity 	:= New_Set_Point;
				Axis_State 			:= Axis_Wait_TGT_Velocity;
			END_IF

			IF Axis_Command 		 = Axis_Emergency_Stop_Request THEN
				Axis_TGT_Position 	:= Axis_Act_Position;
				Axis_TGT_Velocity 	:= 0;
				IF (Axis_Act_Position = Axis_TGT_Position AND Axis_Act_Velocity = Axis_TGT_Velocity) THEN
					Axis_In_Pos 	:= TRUE;
					Axis_In_Vel 	:= TRUE;
					Axis_State 		:= Axis_Check_Command;
				END_IF
			END_IF

		Axis_Wait_TGT_Position:

			IF (Axis_Act_Position = New_Set_Point AND Axis_TGT_Sensor) THEN
				Axis_In_Pos 	:= TRUE;
				Axis_State 		:= Axis_Check_Command;
			END_IF

			Axis_Timer := Axis_Timer - 1;

			IF Axis_Timer = 0 THEN
				Axis_Dev_Fault 	:= TRUE;
				Axis_State 		:= Axis_Fault_State;
			END_IF

		Axis_Wait_TGT_Velocity:

			IF Axis_Act_Velocity = New_Set_Point THEN
				Axis_In_Vel 	:= TRUE;
				Axis_State 		:= Axis_Check_Command;
			END_IF

			Axis_Timer := Axis_Timer - 1;

			IF Axis_Timer = 0 THEN
				Axis_Dev_Fault 	:= TRUE;
				Axis_State 		:= Axis_Fault_State;
			END_IF

		Axis_Fault_State:

			IF Axis_Reset THEN
				Axis_Dev_Fault 	:= FALSE;
				Axis_State 		:= Axis_Check_Command;
			END_IF

	END_CASE

END_FUNCTION_BLOCK
```

### Library Logical/Libraries/Gen_Device (IEC)

#### Types.typ - Exported data types
```iecst
TYPE
	DeviceStateType :
		(
		Dev_Disabled_State,
		Dev_Enable_Phase_State,
		Dev_Enabled_State,
		Dev_Disable_Phase_State
		);
END_TYPE
```

#### Constants.var - Exported constants
```iecst
VAR CONSTANT
	Dev_Without_Feedback : INT := 2#01000000;
	Dev_With_Enable_Feedback : INT := 2#00010000;
	Dev_With_Disable_Feedback : INT := 2#00100000;
	Dev_With_Double_Feedback : INT := 2#00110000;
	Dev_With_Single_Actuation : INT := 2#00000001;
	Dev_With_Double_Actuation : INT := 2#00000011;
	Dev_With_DA_No_Retain : INT := 2#00000010;
	Dev_Feedback_Mask : INT := 2#11110000;
	Dev_Actuation_Mask : INT := 2#00001111;
END_VAR
```

#### Gen_Device.fun - Exported functions and function blocks
```iecst
FUNCTION_BLOCK Gen_Device (*Library for all the devices which have BOOL inputs*)
	VAR_INPUT
		Dev_Operation : {REDUND_UNREPLICABLE} INT;
		Dev_Type : {REDUND_UNREPLICABLE} INT;
		Dev_Enabled_Sensor : {REDUND_UNREPLICABLE} BOOL;
		Dev_Disabled_Sensor : {REDUND_UNREPLICABLE} BOOL;
		Dev_Clock : {REDUND_UNREPLICABLE} BOOL;
		Dev_Enable_Time : {REDUND_UNREPLICABLE} INT;
		Dev_Disable_Time : {REDUND_UNREPLICABLE} INT;
		Dev_Diagnose_Enable : {REDUND_UNREPLICABLE} BOOL;
		Dev_Enable_Preset : {REDUND_UNREPLICABLE} BOOL;
		Dev_Enable : {REDUND_UNREPLICABLE} BOOL;
		Dev_Disable : {REDUND_UNREPLICABLE} BOOL;
	END_VAR
	VAR_OUTPUT
		Dev_Enabled : BOOL;
		Dev_Disabled : BOOL;
		Dev_Enabled_Sensor_Fault : BOOL;
		Dev_Disabled_Sensor_Fault : BOOL;
		Dev_Actuator_Fault : BOOL;
		Dev_Fault : BOOL;
		Dev_Not_Initialized : BOOL;
	END_VAR
	VAR_IN_OUT
		Dev_Enable_Request : BOOL;
		Dev_Disable_Request : BOOL;
	END_VAR
	VAR
		Dev_State : {REDUND_UNREPLICABLE} DeviceStateType;
		Dev_Timer : {REDUND_UNREPLICABLE} INT;
		Dev_Timeout : {REDUND_UNREPLICABLE} BOOL;
	END_VAR
	VAR CONSTANT
		INIT : INT := 0;
		RUN : INT := 1;
	END_VAR
END_FUNCTION_BLOCK
```

#### Gen_Device.st
```iecst
FUNCTION_BLOCK Gen_Device

	//Clock Handling

	IF (Dev_Clock AND (Dev_Timer > 0)) THEN
		Dev_Timer := Dev_Timer - 1;
	END_IF

	//Device Initialization Handling

	CASE (Dev_Type AND Dev_Feedback_Mask) OF

		Dev_With_Enable_Feedback:
			Dev_Disabled_Sensor	:= NOT Dev_Enabled_Sensor AND
			((Dev_State 		 = Dev_Disabled_State) OR
			(Dev_State 			 = Dev_Disable_Phase_State AND Dev_Timeout));

			Dev_Disable 		:= NOT Dev_Enable AND
			((Dev_State			 = Dev_Disabled_State) OR
			(Dev_State 			 = Dev_Disable_Phase_State AND Dev_Timeout));

		Dev_With_Disable_Feedback:
			Dev_Enable 		:= NOT Dev_Disable AND
			((Dev_State 		 = Dev_Enabled_State) OR
			(Dev_State 			 = Dev_Enable_Phase_State AND Dev_Timeout));

			Dev_Enabled_Sensor 	:= NOT Dev_Disabled_Sensor AND
			((Dev_State 		 = Dev_Enabled_State) OR
			(Dev_State 			 = Dev_Enable_Phase_State AND Dev_Timeout));

		Dev_Without_Feedback:
			Dev_Enable 		:= (Dev_State = Dev_Enabled_State) OR
			(Dev_State 			 = Dev_Enable_Phase_State AND Dev_Timeout);
			Dev_Disable 		:= (Dev_State = Dev_Disabled_State) OR
			(Dev_State 			 = Dev_Disable_Phase_State AND Dev_Timeout);

			Dev_Enabled_Sensor  := (Dev_State = Dev_Enabled_State) OR
			((Dev_State 		 = Dev_Enable_Phase_State) AND Dev_Timeout);
			Dev_Disabled_Sensor := (Dev_State = Dev_Disabled_State) OR
			((Dev_State			 = Dev_Disable_Phase_State) AND Dev_Timeout);
	END_CASE

	// Device Sensor Handler
	IF (Dev_Operation = INIT) THEN

		CASE (Dev_Type AND Dev_Feedback_Mask) OF
			Dev_With_Enable_Feedback:
				Dev_Disable 	:= NOT Dev_Enable;

			Dev_With_Disable_Feedback:
				Dev_Enable 	:=  NOT Dev_Disable;

			Dev_Without_Feedback:
				Dev_Enable 	:= Dev_Enable_Preset;
				Dev_Disable 	:= NOT Dev_Enable;
		END_CASE

		Dev_Enable_Request 		:= FALSE;
		Dev_Disable_Request 	:= FALSE;
		IF (Dev_Enable_Preset) THEN
			Dev_Enabled 			:= TRUE;
			Dev_Timer 			:= Dev_Enable_Time;
			IF NOT (Dev_Disable AND Dev_Enable) THEN
				Dev_State 		:= Dev_Enable_Phase_State;
			ELSE
				Dev_State 		:= Dev_Enabled_State;
			END_IF
			Dev_Not_Initialized := NOT Dev_Enable OR Dev_Disable;

		ELSE
			Dev_Enabled			:= FALSE;
			Dev_Timer 			:= Dev_Disable_Time;
			IF NOT (Dev_Disable AND Dev_Enable) THEN
				Dev_State 		:= Dev_Disable_Phase_State;
			ELSE
				Dev_State 		:= Dev_Disabled_State;
			END_IF
			Dev_Not_Initialized := (Dev_Enable OR NOT Dev_Disable);

		END_IF
	END_IF

	// Device Control Handling

	CASE (Dev_State) OF

		Dev_Disabled_State:
			Dev_Disable_Request := FALSE;
			IF Dev_Enable_Request THEN
				Dev_Enabled 		:= TRUE;
				Dev_Timer 		:= Dev_Enable_Time;
				Dev_State 		:= Dev_Enable_Phase_State;
			END_IF

		Dev_Enable_Phase_State:
			IF Dev_Disable_Request THEN
				Dev_Enable_Request 	:= FALSE;
				Dev_Enabled 			:= FALSE;
				Dev_Timer 			:= Dev_Disable_Time;
				Dev_State 			:= Dev_Disable_Phase_State;
			END_IF

			IF Dev_Enabled_Sensor THEN
				Dev_Enable_Request 	:= FALSE;
				Dev_Timer 			:= 0;
				Dev_State 			:= Dev_Enabled_State;
			END_IF

		Dev_Enabled_State:
			Dev_Enable_Request	:= FALSE;
			IF Dev_Disable_Request THEN
				Dev_Enabled 		:= FALSE;
				Dev_Timer 		:= Dev_Disable_Time;
				Dev_State 		:= Dev_Disable_Phase_State;
			END_IF

		Dev_Disable_Phase_State:
			IF Dev_Enable_Request THEN
				Dev_Disable_Request := FALSE;
				Dev_Enabled 			:= TRUE;
				Dev_Timer 			:= Dev_Enable_Time;
				Dev_State 			:= Dev_Enable_Phase_State;
			END_IF

			IF Dev_Disabled_Sensor THEN
				Dev_Disable_Request := FALSE;
				Dev_Timer 			:= 0;
				Dev_State 			:= Dev_Disabled_State;
			END_IF
	END_CASE

	// Device Diagnostic Handling

	Dev_Timeout 				:= (Dev_Timer = 0);
	Dev_Disabled_Sensor_Fault 	:= ((NOT Dev_Enabled AND NOT Dev_Disabled_Sensor AND NOT Dev_Enabled_Sensor) OR (Dev_Enabled AND Dev_Disabled_Sensor AND Dev_Enabled_Sensor)) AND Dev_Timeout;
	Dev_Enabled_Sensor_Fault 	:= ((NOT Dev_Enabled AND Dev_Disabled_Sensor AND Dev_Enabled_Sensor) OR (Dev_Enabled AND NOT Dev_Disabled_Sensor AND NOT Dev_Enabled_Sensor)) AND Dev_Timeout;
	Dev_Actuator_Fault 			:= ((NOT Dev_Enabled AND NOT Dev_Disabled_Sensor AND Dev_Enabled_Sensor) OR (Dev_Enabled AND Dev_Disabled_Sensor AND NOT Dev_Enabled_Sensor)) AND Dev_Timeout;
	Dev_Fault 					:= Dev_Disabled_Sensor_Fault OR Dev_Enabled_Sensor_Fault OR Dev_Actuator_Fault;

	// Device Actuators Handling

	CASE (Dev_Type AND Dev_Actuation_Mask) OF

		Dev_With_Double_Actuation:
			Dev_Disabled := NOT Dev_Enabled;

		Dev_With_DA_No_Retain:
			Dev_Enabled 	:= Dev_Enabled AND (Dev_State = Dev_Enable_Phase_State);
			Dev_Disabled := NOT Dev_Enabled AND (Dev_State = Dev_Disable_Phase_State);

	END_CASE

END_FUNCTION_BLOCK
```

### Library Logical/Libraries/Blink (IEC)

#### Blink.fun - Exported functions and function blocks
```iecst
FUNCTION_BLOCK Blink
	VAR_INPUT
		LED_State : STRING[80];
	END_VAR
	VAR_OUTPUT
		LED_Light : BOOL;
	END_VAR
	VAR
		Timer : TON;
		State : INT := 0;
	END_VAR
END_FUNCTION_BLOCK
```

#### Blink.st
```iecst
(* For Turning LED ON/OFF/Blink *)
FUNCTION_BLOCK Blink

	IF LED_State = 'on' THEN
		LED_Light := TRUE;
	END_IF

	IF LED_State = 'off' THEN
		LED_Light := FALSE;
	END_IF

	IF LED_State = 'blink' THEN

		CASE State OF

			0:
				Timer(IN := TRUE, PT := T#500ms);
				IF Timer.Q = TRUE THEN
					Timer(IN 	:= FALSE);
					LED_Light 	:= TRUE;
					State 		:= 1;
				END_IF

			1:
				Timer(IN := TRUE, PT := T#500ms);
				IF Timer.Q = TRUE THEN
					Timer(IN 	:= FALSE);
					LED_Light 	:= FALSE;
					State 		:= 0;
				END_IF
		END_CASE

	END_IF

END_FUNCTION_BLOCK
```

- Visualisation Logical/mappView (not shown)

### Program Logical/Input_Bridge (IEC)

#### Variables.var
```iecst
VAR
	IR_Sensor_1 : S_filter; (*laser_sensor_IR*)
	IR_Sensor_2 : S_filter; (*laser_sensor2_IR*)
	CarriageB : S_filter; (*carriage_2_AXIS*)
	Carriage : S_filter; (*carriage_2_AXIS*)
	Pusher_1_B : S_filter; (*pusher_LBK*)
	Pusher_1_F : S_filter; (*pusher_LFR*)
	Turn_Push_B : S_filter; (*turnpusher_LBK*)
	Turn_Push_F : S_filter; (*turnpusher_LFR*)
	Gantry_Crane : S_filter; (*gantry_crane_AXIS*)
	Box_Crane : S_filter; (*box_crane_AXIS*)
	Vacuum : S_filter; (*vacuum_box_crane_VACUUM*)
	Pallet_lift : S_filter; (*pallet_lifter_AXIS*)
	Pallet_holder : S_filter; (*pallet_fork_left_FB*)
	IR_Sensor_3 : S_filter; (*pallet_light_barrier_1_IR*)
	IR_Sensor_4 : S_filter; (*pallet_light_barrier_2_IR*)
END_VAR
```

#### Main.st
```iecst
PROGRAM _INIT
	(* Insert code here *)

END_PROGRAM

PROGRAM _CYCLIC
	// Feeder Input Variables
	IR_Sensor_1(Sensor_Raw 	:= ComTCP_SimInputs.laser_sensor_IR,
				threshold_B := 10,
				Is_Bool 	:= TRUE);
	IR_Sensor_2(Sensor_Raw 	:= ComTCP_SimInputs.laser_sensor2_IR,
				threshold_B := 2,
				Is_Bool 	:= TRUE);
	Carriage(	Sensor_Data := ComTCP_SimInputs.carriage_2_AXIS,
				threshold_F := 0.8,
				Is_Bool 	:= FALSE);
	CarriageB(	Sensor_Raw 	:= ComTCP_SimInputs.carriage_2_RCHD,
				threshold_B := 10,
				Is_Bool 	:= TRUE);
	Pusher_1_B( Sensor_Raw 	:= ComTCP_SimInputs.pusher_LBK,
				threshold_B := 10,
				Is_Bool 	:= TRUE);
	Pusher_1_F(	Sensor_Raw 	:= ComTCP_SimInputs.pusher_LFR,
				threshold_B := 10,
				Is_Bool 	:= TRUE);
	Turn_Push_B(Sensor_Raw 	:= ComTCP_SimInputs.turnpusher_LBK,
				threshold_B := 10,
				Is_Bool 	:= TRUE);
	Turn_Push_F(Sensor_Raw 	:= ComTCP_SimInputs.turnpusher_LFR,
				threshold_B := 10,
				Is_Bool 	:= TRUE);

	//Filtered Data
	I_IR_Sensor_1 			:= IR_Sensor_1.Sensor_Filtered; //First Laser Sensor;
	I_IR_Sensor_2 			:= IR_Sensor_2.Sensor_Filtered; //Second Leser Sensor;
	I_Carriage_Push_Act_Pos := Carriage.Sensor_Data_Filtered; //Actual postion of Group box pusher;
	I_Carriage_Push_Tar_Rec := CarriageB.Sensor_Filtered; //Group box reached target;
	I_Pusher_1_B 			:= Pusher_1_B.Sensor_Filtered; //Pusher 1 Back Position;
	I_Pusher_1_F 			:= Pusher_1_F.Sensor_Filtered; //Pusher 1 Front Position;
	I_Turn_Push_B 			:= Turn_Push_B.Sensor_Filtered; //Turn Pusher back position;
	I_Turn_Push_F 			:= Turn_Push_F.Sensor_Filtered; //Turn Pusher Front position;

	//Crane Input Variables
	Gantry_Crane(	Sensor_Data := ComTCP_SimInputs.gantry_crane_AXIS,
					threshold_F := 0.99,
					Is_Bool 	:= FALSE);
	Box_Crane(		Sensor_Data := ComTCP_SimInputs.box_crane_AXIS,
					threshold_F := 0.99,
					Is_Bool 	:= FALSE);
	Vacuum(			Sensor_Raw 	:= ComTCP_SimInputs.vaccum_box_crane_VACUUM,
					threshold_B := 10,
					Is_Bool 	:= TRUE);
	//Filtered Data
	I_Gantry_Crane_Act_Pos 		:= Gantry_Crane.Sensor_Data_Filtered; //Gantry Crane Actual Position;
	I_Box_Crane_Act_Pos 		:= Box_Crane.Sensor_Data_Filtered; // Box Crane Actual Position;
	I_Vacuum_retention_act 		:= Vacuum.Sensor_Filtered; //Vacuum capfor cartboard retention active;

	//Pallet Handler Input Variables
	Pallet_lift(	Sensor_Data := ComTCP_SimInputs.pallet_lifter_AXIS,
					threshold_F := 0.8,
					Is_Bool 	:= FALSE);
	Pallet_holder(	Sensor_Raw 	:= ComTCP_SimInputs.pallet_fork_left_FB,
					threshold_B := 10,
					Is_Bool 	:= TRUE);
	IR_Sensor_3(	Sensor_Raw 	:= ComTCP_SimInputs.pallet_light_barrier_1_IR,
					threshold_B := 1,
					Is_Bool 	:= TRUE);
	IR_Sensor_4(	Sensor_Raw 	:= ComTCP_SimInputs.pallet_light_barrier_2_IR,
					threshold_B := 1,
					Is_Bool 	:= TRUE);
	//Filtered Data
	I_Pallet_lift_Act_Pos 		:= Pallet_lift.Sensor_Data_Filtered; //Pallet lifter actual position;
	I_Pallet_holder_State 		:= Pallet_holder.Sensor_Filtered; //pallet fork open;
	I_IR_Sensor_3 				:= IR_Sensor_3.Sensor_Filtered; //pallet present before assembly;
	I_IR_Sensor_4 				:= IR_Sensor_4.Sensor_Filtered; //pallet present after assembly;

	//HMI Main Input parameters
	Service_Mode := Service_Mode_HMI;
END_PROGRAM

PROGRAM _EXIT
	(* Insert code here *)

END_PROGRAM
```

### Program Logical/Output_Bridge (IEC)

#### Main.st
```iecst
PROGRAM _INIT
	(* Insert code here *)

END_PROGRAM

PROGRAM _CYCLIC
	// Feeder Output Variables
	ComTCP_SimOutputs.conveyor_if_FWD 			:= O_Conveyor_1; //Conveyor_if control
	ComTCP_SimOutputs.pusher_FW 				:= O_Pusher_1; //pusher control
	ComTCP_SimOutputs.conveyer_turn1_FWD 		:= O_Conveyor_2; //conveyor_turn1 control
	ComTCP_SimOutputs.conveyer_end_FWD 			:= O_Conveyor_3; //conveyor_end control
	ComTCP_SimOutputs.turnpusher_FWD 			:= O_Turn_Pusher_ON; //turnpusher Forward
	ComTCP_SimOutputs.turnpusher_BWD 			:= O_Turn_Pusher_OFF; //turnpusher Backward
	ComTCP_SimOutputs.carriage_2_TGT_POS		:= O_Carriage_Tar_Pos; //Set Target Position for carriage

	//Crane Output Variables
	ComTCP_SimOutputs.gantry_crane_TGT_POS 		:= O_Gantry_Crane_Tar_Pos; //Set Gantry Crane Target Position
	ComTCP_SimOutputs.box_crane_TGT_POS 		:= O_Box_Crane_Tar_Pos; //Set Box Crane Target Position
	ComTCP_SimOutputs.cartboard_TRIG 			:= O_Cartboard_Trig; //release of first cartboard in the pile.
	ComTCP_SimOutputs.vaccum_box_crane_GRIP 	:= O_Vacuum_Grip_act; //holding the cartboard using vaccum
	ComTCP_SimOutputs.slide_rail_right_EN 		:= O_Box_Holder; //Hold box during the crane motion
	ComTCP_SimOutputs.pusher_z_EN 				:= O_Pusher_z; // move down layer pusher
	ComTCP_SimOutputs.pusher_x_EN 				:= O_Pusher_x; //move forward layer pusher

	//Pallet Handler Output Variables
	ComTCP_SimOutputs.pallet_lifter_TGT_POS 	:= O_Pallet_lift_Tar_Pos; //pallet lifter target position;
	ComTCP_SimOutputs.pallet_fork_left_EN 		:= O_Pallet_Holder; //Command to open fork;
	ComTCP_SimOutputs.pallet_conveyor_1_FWD 	:= O_Conveyor_4; //Controlling Pallet Conveyor 4;
	ComTCP_SimOutputs.pallet_conveyor_2_ACT_VEL := O_Conveyor_5_vel; //Controlling Pallet Conveyor 5 with velocity;

END_PROGRAM

PROGRAM _EXIT
	(* Insert code here *)

END_PROGRAM
```

### Program Logical/Main_Control (IEC)

#### Types.typ
```iecst
TYPE
	States :
		(
		Emergency_Stop_Seq := 1,
		Stop_Seq := 2,
		Wait_For_Restart := 3,
		Wait_Start := 4,
		Box_In_Position := 5,
		Box_On_The_Crane := 6,
		Wait_For_Pallet := 7,
		Box_On_The_Pallet := 8,
		Pallet_Exit := 9
		);
END_TYPE
```

#### Variables.var
```iecst
VAR
	Main_State : States := Wait_Start;
	Restart_Req : BOOL := FALSE;
	Old_State : States;
	Immediate_Stop_Req : BOOL := FALSE;
	On_Phase_Stop_Req : BOOL := FALSE;
	Stop_Request : BOOL := FALSE;
	New_Variable : USINT;
END_VAR
```

#### Main.st
```iecst
PROGRAM _INIT
	(* Insert code here *)

END_PROGRAM

PROGRAM _CYCLIC
	(* Insert code here *)

	CASE Main_State OF
		Emergency_Stop_Seq:
			M_Current_State := 'Emergency Stop Sequence';
			En_Machine 		:= FALSE;
			Start_Machine 	:= FALSE;
			IF (NOT Emergency_Stop AND NOT F_Emergency_Stop AND NOT C_Emergency_Stop AND NOT P_Emergency_Stop) THEN
				F_Reset_Config 	:= TRUE;
				C_Reset_Config 	:= TRUE;
				P_Reset_Config 	:= TRUE;
				Restart_Req 	:= FALSE;
				Main_State 		:= Wait_Start;
			END_IF

		Stop_Seq:
			M_Current_State := 'Stop Sequence';
			En_Machine 		:= FALSE;
			Start_Machine 	:= FALSE;
			Stop_Request 	:= TRUE;
			IF( NOT Immediate_Stop AND NOT F_Immediate_Stop AND NOT C_Immediate_Stop AND NOT P_Immediate_Stop) AND (NOT On_Phase_Stop AND NOT F_On_Phase_Stop AND NOT C_On_Phase_Stop AND NOT P_On_Phase_Stop) THEN
				En_Machine 	:= TRUE;
				Restart_Req := TRUE;
				Main_State 	:= Wait_Start;
			END_IF

			IF Emergency_Stop AND (On_Phase_Stop_Req OR Immediate_Stop_Req) THEN
				On_Phase_Stop_Req 	:= FALSE;
				Immediate_Stop_Req 	:= FALSE;
				F_Immediate_Stop 	:= FALSE;
				F_On_Phase_Stop 	:= FALSE;
				C_Immediate_Stop 	:= FALSE;
				C_On_Phase_Stop 	:= FALSE;
				P_Immediate_Stop 	:= FALSE;
				P_On_Phase_Stop 	:= FALSE;
				Main_State 			:= Wait_Start;
			END_IF

			IF Immediate_Stop AND On_Phase_Stop_Req THEN
				On_Phase_Stop_Req 	:= FALSE;
				F_On_Phase_Stop 	:= FALSE;
				C_On_Phase_Stop 	:= FALSE;
				P_On_Phase_Stop 	:= FALSE;
				Main_State 			:= Wait_Start;
			END_IF

		Wait_For_Restart:
			M_Current_State := 'Wait For Restart';
			IF (NOT F_Restart AND NOT C_Restart AND NOT P_Restart) THEN
				Stop_Request 		:= FALSE;
				Restart_Req 	:= FALSE;
				Start_Feeder 	:= TRUE;
				Start_Crane 	:= TRUE;
				Start_Pallet 	:= TRUE;
				Main_State 		:= Old_State;
			END_IF

		Wait_Start:
			M_Current_State := 'Wait Start';
			IF (Start_Machine AND En_Machine AND Restart_Req) THEN
				F_Restart 	:= TRUE;
				C_Restart 	:= TRUE;
				P_Restart 	:= TRUE;
				Main_State 	:= Wait_For_Restart;
			END_IF

			IF (NOT F_Reset_Config AND NOT C_Reset_Config AND NOT P_Reset_Config) THEN
				En_Machine := TRUE;
			END_IF

			IF (Start_Machine AND En_Machine AND NOT Restart_Req) THEN
				Start_Feeder 	:= TRUE;
				Start_Crane 	:= TRUE;
				Start_Pallet 	:= TRUE;
				Main_State 		:= Box_In_Position;
			END_IF

			IF Emergency_Stop THEN
				F_Emergency_Stop 	:= TRUE;
				C_Emergency_Stop 	:= TRUE;
				P_Emergency_Stop 	:= TRUE;
				Main_State 			:= Emergency_Stop_Seq;
			END_IF

			IF Immediate_Stop THEN
				Immediate_Stop_Req 	:= TRUE;
				IF NOT Stop_Request THEN
					Old_State 		:= Main_State;
				END_IF
				F_Immediate_Stop 	:= TRUE;
				C_Immediate_Stop 	:= TRUE;
				P_Immediate_Stop 	:= TRUE;
				Main_State := Stop_Seq;
			END_IF

			IF On_Phase_Stop AND NOT Stop_Request THEN
				On_Phase_Stop_Req := TRUE;
				IF NOT Stop_Request THEN
					Old_State := Main_State;
				END_IF
				F_On_Phase_Stop 	:= TRUE;
				C_On_Phase_Stop 	:= TRUE;
				P_On_Phase_Stop 	:= TRUE;
				Main_State 			:= Stop_Seq;
			END_IF

		Box_In_Position:
			M_Current_State := 'Box In Position';
			P_Exit_Done 	:= FALSE;
			Boxes_On_The_P 	:= FALSE;
			IF (F_Ready AND C_Ready) THEN
				Load_Boxes_On_The_C := TRUE;
				Main_State 			:= Box_On_The_Crane;
			END_IF

			IF Emergency_Stop THEN
				F_Emergency_Stop 	:= TRUE;
				C_Emergency_Stop 	:= TRUE;
				P_Emergency_Stop 	:= TRUE;
				Main_State 			:= Emergency_Stop_Seq;
			END_IF

			IF Immediate_Stop THEN
				Immediate_Stop_Req 	:= TRUE;
				Old_State 			:= Main_State;
				F_Immediate_Stop 	:= TRUE;
				C_Immediate_Stop 	:= TRUE;
				P_Immediate_Stop 	:= TRUE;
				Main_State := Stop_Seq;
			END_IF

			IF On_Phase_Stop THEN
				On_Phase_Stop_Req 	:= TRUE;
				Old_State 			:= Main_State;
				F_On_Phase_Stop 	:= TRUE;
				C_On_Phase_Stop 	:= TRUE;
				P_On_Phase_Stop 	:= TRUE;
				Main_State 			:= Stop_Seq;
			END_IF

		Box_On_The_Crane:
			M_Current_State := 'Box On The Crane';
			IF Boxes_On_The_C THEN
				F_Ready 			:= FALSE;
				C_Ready 			:= FALSE;
				Load_Boxes_On_The_C := FALSE;
				Hold_Boxes 			:= TRUE;
				Main_State 			:= Wait_For_Pallet;
			END_IF

			IF Emergency_Stop THEN
				F_Emergency_Stop 	:= TRUE;
				C_Emergency_Stop 	:= TRUE;
				P_Emergency_Stop 	:= TRUE;
				Main_State 			:= Emergency_Stop_Seq;
			END_IF

			IF Immediate_Stop THEN
				Immediate_Stop_Req 	:= TRUE;
				Old_State 			:= Main_State;
				F_Immediate_Stop 	:= TRUE;
				C_Immediate_Stop 	:= TRUE;
				P_Immediate_Stop 	:= TRUE;
				Main_State 			:= Stop_Seq;
			END_IF

			IF On_Phase_Stop THEN
				On_Phase_Stop_Req 	:= TRUE;
				Old_State 			:= Main_State;
				F_On_Phase_Stop 	:= TRUE;
				C_On_Phase_Stop 	:= TRUE;
				P_On_Phase_Stop 	:= TRUE;
				Main_State 			:= Stop_Seq;
			END_IF

		Wait_For_Pallet:
			M_Current_State := 'Wait For Pallet';
			IF P_Ready THEN
				Boxes_On_The_C 		:= FALSE;
				Load_Boxes_On_The_P := TRUE;
				Main_State 			:= Box_On_The_Pallet;
			END_IF

			IF Emergency_Stop THEN
				F_Emergency_Stop 	:= TRUE;
				C_Emergency_Stop 	:= TRUE;
				P_Emergency_Stop 	:= TRUE;
				Main_State 			:= Emergency_Stop_Seq;
			END_IF

			IF Immediate_Stop THEN
				Immediate_Stop_Req 	:= TRUE;
				Old_State 			:= Main_State;
				F_Immediate_Stop 	:= TRUE;
				C_Immediate_Stop 	:= TRUE;
				P_Immediate_Stop 	:= TRUE;
				Main_State 			:= Stop_Seq;
			END_IF

			IF On_Phase_Stop THEN
				On_Phase_Stop_Req 	:= TRUE;
				Old_State 			:= Main_State;
				F_On_Phase_Stop 	:= TRUE;
				C_On_Phase_Stop 	:= TRUE;
				P_On_Phase_Stop 	:= TRUE;
				Main_State 			:= Stop_Seq;
			END_IF

		Box_On_The_Pallet:
			M_Current_State := 'Box On The Pallet';
			IF Boxes_On_The_P THEN
				Hold_Boxes 			:= FALSE;
				Load_Boxes_On_The_P := FALSE;
				IF Second_Layer THEN
					P_Exit_En 	:= TRUE;
					Main_State 	:= Pallet_Exit;
				END_IF
				IF NOT Second_Layer THEN
					Main_State 	:= Wait_Start;
				END_IF
			END_IF

			IF Emergency_Stop THEN
				F_Emergency_Stop 	:= TRUE;
				C_Emergency_Stop 	:= TRUE;
				P_Emergency_Stop 	:= TRUE;
				Main_State 			:= Emergency_Stop_Seq;
			END_IF

			IF Immediate_Stop THEN
				Immediate_Stop_Req 	:= TRUE;
				Old_State 			:= Main_State;
				F_Immediate_Stop 	:= TRUE;
				C_Immediate_Stop 	:= TRUE;
				P_Immediate_Stop 	:= TRUE;
				Main_State 			:= Stop_Seq;
			END_IF

			IF On_Phase_Stop THEN
				On_Phase_Stop_Req 	:= TRUE;
				Old_State 			:= Main_State;
				F_On_Phase_Stop 	:= TRUE;
				C_On_Phase_Stop 	:= TRUE;
				P_On_Phase_Stop 	:= TRUE;
				Main_State 			:= Stop_Seq;
			END_IF

		Pallet_Exit:
			M_Current_State := 'Pallet Exit';
			IF P_Exit_Done THEN
				P_Ready 		:= FALSE;
				P_Exit_En 		:= FALSE;
				Second_Layer 	:= FALSE;
				Main_State 		:= Wait_Start;
			END_IF

			IF Emergency_Stop THEN
				F_Emergency_Stop 	:= TRUE;
				C_Emergency_Stop 	:= TRUE;
				P_Emergency_Stop 	:= TRUE;
				Main_State 			:= Emergency_Stop_Seq;
			END_IF

			IF Immediate_Stop THEN
				Immediate_Stop_Req 	:= TRUE;
				Old_State 			:= Main_State;
				F_Immediate_Stop 	:= TRUE;
				C_Immediate_Stop 	:= TRUE;
				P_Immediate_Stop 	:= TRUE;
				Main_State 			:= Stop_Seq;
			END_IF

			IF On_Phase_Stop THEN
				On_Phase_Stop_Req 	:= TRUE;
				Old_State 			:= Main_State;
				F_On_Phase_Stop 	:= TRUE;
				C_On_Phase_Stop 	:= TRUE;
				P_On_Phase_Stop 	:= TRUE;
				Main_State 			:= Stop_Seq;
			END_IF

	END_CASE

END_PROGRAM

PROGRAM _EXIT
	(* Insert code here *)

END_PROGRAM
```

### Program Logical/Feeder (IEC)

#### Types.typ
```iecst
TYPE
	Feeder_State :
		(
		Feeder_Stop_Seq := 1,
		Feeder_Stop_Done := 2,
		Reset_Feeder_Config := 3,
		Restore_Feeder_Config_1 := 4,
		Restore_Feeder_Config_2 := 5,
		Restore_Feeder_Config_3 := 6,
		Wait_Start := 7,
		Wait_Conveyor_1_Active := 8,
		Wait_Pusher_Position := 9,
		Layer_Check := 10,
		Line_Check := 11,
		Wait_IR_Sensor_2 := 12,
		Box_In_Pos := 13,
		Wait_Conveyor_Stop := 14,
		Feeder_Idle := 15,
		Carriage_FWD_Pos := 16,
		Carriage_BWD_Pos := 17,
		Wait_Start_Pos := 18
		);
END_TYPE
```

#### Variables.var
```iecst
VAR
	State : INT := 0;
	Feeder_Current_State : Feeder_State := Wait_Start;
END_VAR
(*First Conveyor (Conveyor_if)*)
VAR
	Conveyor_1 : Gen_Device;
	Conv_1_En_Time : INT := 20;
	Conv_1_Dis_Time : INT := 20;
END_VAR
(*Pusher*)
VAR
	Pusher_1 : Gen_Device;
	Pusher_1_En_Time : INT := 60;
	Pusher_1_Dis_Time : INT := 60;
END_VAR
(*Second Conveyor (Conveyor_turn1)*)
VAR
	Conveyor_2 : Gen_Device;
	Conv_2_En_Time : INT := 20;
	Conv_2_Dis_Time : INT := 20;
END_VAR
(*Third Conveyor (Conveyor_end)*)
VAR
	Conveyor_3 : Gen_Device;
	Conv_3_En_Time : INT := 20;
	Conv_3_Dis_Time : INT := 20;
END_VAR
(*Turn Pusher*)
VAR
	Turn_Pusher : Gen_Device;
	Turn_Pusher_En_Time : INT := 60;
	Turn_Pusher_Dis_Time : INT := 60;
END_VAR
(*Carriage*)
VAR
	Carriage : Gen_Axis;
	Carriage_Pos_Reached : BOOL;
	Carriage_Tar_Pos : REAL;
	Main_Line : BOOL := FALSE;
END_VAR
(*Faults*)
VAR
	Feeder_Old_State : Feeder_State;
	En_Dis_Array : ARRAY[0..9] OF BOOL := [10(FALSE)];
	Old_Pos : REAL;
	a : INT := 0;
	End_Layer : BOOL := FALSE;
	En_Dis_Counter : INT;
	Sensor_Reached : ARRAY[0..1] OF BOOL := [2(FALSE)];
	Carriage_Pos_Restored : BOOL := FALSE;
	Check_Pos : BOOL := FALSE;
	Sensor_Memory : ARRAY[0..1] OF BOOL := [2(FALSE)];
	Stop_Request : BOOL := FALSE;
END_VAR
VAR CONSTANT
	Idle : WORD := 0;
	Change_Vel : WORD := 1;
	Change_Pos : WORD := 2;
	Emergency_Stop_Req : WORD := 3;
END_VAR
VAR
	Conv_1_dis_req : BOOL;
	Conv_2_dis_req : BOOL;
	Pusher_dis_req : BOOL;
	Conv_3_dis_req : BOOL;
	Turnpusher_dis_req : BOOL;
	Conv_1_en_req : BOOL;
	Conv_2_en_req : BOOL;
	Pusher_en_req : BOOL;
	Conv_3_en_req : BOOL;
	Turnpusher_en_req : BOOL;
	New_Variable6 : USINT;
	New_Variable5 : USINT;
	New_Variable4 : USINT;
	New_Variable3 : USINT;
	New_Variable2 : USINT;
	New_Variable1 : USINT;
	New_Variable : USINT;
END_VAR
```

#### Main.st
```iecst
PROGRAM _INIT
	(* Insert code here *)

END_PROGRAM

PROGRAM _CYCLIC
	(* Insert code here *)
	CASE State OF
		0: //
			IF Service_Mode THEN
				State := 1;
			END_IF

			CASE Feeder_Current_State OF

				Feeder_Stop_Seq:
					F_Current_State			:= 'Feeder Stop Sequence';
					Start_Feeder 			:= FALSE;
					Conv_1_dis_req 			:= TRUE;
					Conv_2_dis_req 			:= TRUE;
					Conv_3_dis_req 			:= TRUE;
					Carriage.Axis_Command 	:= Emergency_Stop_Req;
					Feeder_Current_State 	:= Feeder_Stop_Done;

				Feeder_Stop_Done:
					F_Current_State			:= 'Feeder Stop Done';
					IF (NOT Conv_1_dis_req AND NOT Conv_2_dis_req AND NOT Conv_3_dis_req AND Carriage_Pos_Reached)THEN
						Carriage.Axis_Command 	:= Idle;
						F_Emergency_Stop 		:= FALSE;
						F_Immediate_Stop 		:= FALSE;
						F_On_Phase_Stop 		:= FALSE;
						Stop_Request 			:= TRUE;
						Feeder_Current_State 	:= Wait_Start;
					END_IF

				Reset_Feeder_Config:
					F_Current_State	:= 'Reset Feeder Configuration';
					IF NOT F_Reset_Config THEN
						Feeder_Current_State 	:= Wait_Start;
					END_IF

					IF (Carriage_Pos_Reached AND NOT Pusher_dis_req AND NOT Turnpusher_dis_req) THEN
						Carriage.Axis_Command 	:= Idle;
						Sensor_Memory[0] 		:= FALSE;
						Sensor_Memory[1] 		:= FALSE;
						Sensor_Reached[0] 		:= FALSE;
						Sensor_Reached[1] 		:= FALSE;
						FOR a := 0 TO 9 DO
							En_Dis_Array[a] 	:= FALSE;
						END_FOR
						F_Reset_Config			:= FALSE;
						Feeder_Current_State 	:= Wait_Start;
					END_IF

				Restore_Feeder_Config_1:
					F_Current_State			:= 'Restore Feeder Configuration 1';
					Carriage.Axis_Command 	:= Idle;
					FOR a := 0 TO 9 DO
						IF En_Dis_Array[a] THEN
							CASE a OF
								0:
									Conv_1_en_req 		:= TRUE;
								1:
									Conv_1_dis_req 		:= TRUE;
								2:
									Conv_2_en_req 		:= TRUE;
								3:
									Conv_2_dis_req 		:= TRUE;
								4:
									Conv_3_en_req 		:= TRUE;
								5:
									Conv_3_dis_req 		:= TRUE;
								6:
									Pusher_en_req 		:= TRUE;
								7:
									Pusher_dis_req 		:= TRUE;
								8:
									Turnpusher_en_req 	:= TRUE;
								9:
									Turnpusher_dis_req 	:= TRUE;

							END_CASE
						END_IF
					END_FOR
					En_Dis_Counter 			:= 70;
					Feeder_Current_State 	:= Restore_Feeder_Config_2;

				Restore_Feeder_Config_2:
					F_Current_State	:= 'Restore Feeder Configuration 2';
					FOR a := 0 TO 9 DO
						IF En_Dis_Array[a] THEN
							CASE a OF
								0:
									IF NOT Conv_1_en_req THEN
										En_Dis_Array [a] := TRUE;
									END_IF

								1:
									IF NOT Conv_1_dis_req THEN
										En_Dis_Array [a] := TRUE;
									END_IF

								2:
									IF NOT Conv_2_en_req THEN
										En_Dis_Array [a] := TRUE;
									END_IF

								3:
									IF NOT Conv_2_dis_req THEN
										En_Dis_Array [a] := TRUE;
									END_IF

								4:
									IF NOT Conv_3_en_req THEN
										En_Dis_Array [a] := TRUE;
									END_IF

								5:
									IF NOT Conv_3_dis_req THEN
										En_Dis_Array [a] := TRUE;
									END_IF

								6:
									IF NOT Pusher_en_req THEN
										En_Dis_Array [a] := TRUE;
									END_IF

								7:
									IF NOT Pusher_dis_req THEN
										En_Dis_Array [a] := TRUE;
									END_IF

								8:
									IF NOT Turnpusher_en_req THEN
										En_Dis_Array [a] := TRUE;
									END_IF

								9:
									IF NOT Turnpusher_dis_req THEN
										En_Dis_Array [a] := TRUE;
									END_IF
							END_CASE
						END_IF
					END_FOR

					En_Dis_Counter := En_Dis_Counter - 1;

					IF En_Dis_Counter = 0 THEN
						IF Check_Pos THEN
							Carriage_Tar_Pos 		:= Old_Pos;
							Carriage.Axis_Command 	:= Change_Pos;
						END_IF
						Feeder_Current_State 		:= Restore_Feeder_Config_3;
					END_IF

				Restore_Feeder_Config_3:
					F_Current_State	:= 'Restore Feeder Configuration 3';
					IF (Carriage_Pos_Reached AND Check_Pos) THEN
						Carriage.Axis_Command := Idle;
						Carriage_Pos_Restored := TRUE;
					END_IF
					IF (NOT Check_Pos OR Carriage_Pos_Restored) THEN
						Stop_Request				:= FALSE;
						F_Restart 				:= FALSE;
						Feeder_Current_State 	:= Feeder_Old_State;
					END_IF

				Wait_Start:
					F_Current_State	:= 'Wait Start';
					IF F_Restart THEN
						Feeder_Current_State 	:= Restore_Feeder_Config_1;
					END_IF

					IF F_Reset_Config THEN
						Box_Counter 			:= 0;
						F_Ready 				:= FALSE;
						C_Layer_Counter 		:= FALSE;
						Second_Layer 			:= FALSE;
						Load_Boxes_On_The_C 	:= FALSE;
						Boxes_On_The_C 			:= FALSE;
						Pusher_dis_req 			:= TRUE;
						Turnpusher_dis_req 		:= TRUE;
						Carriage_Tar_Pos 		:= 0;
						Carriage.Axis_Command 	:= Change_Pos;
						Feeder_Current_State 	:= Reset_Feeder_Config;
					END_IF

					IF (Start_Feeder AND NOT F_Reset_Config AND NOT F_Restart) THEN
						Conv_1_en_req 			:= TRUE;
						Feeder_Current_State 	:= Wait_Conveyor_1_Active;
					END_IF

					IF F_Emergency_Stop THEN
						Feeder_Current_State 	:= Feeder_Stop_Seq;
					END_IF

					IF F_Immediate_Stop AND NOT Stop_Request THEN
						Feeder_Old_State 		:= Feeder_Current_State;
						Feeder_Current_State 	:= Feeder_Stop_Seq;
					END_IF

					IF F_Immediate_Stop AND Stop_Request THEN
						Feeder_Current_State 	:= Feeder_Stop_Seq;
					END_IF

				Wait_Conveyor_1_Active:
					F_Current_State	:= 'Wait Conveyor 1 Active';
					IF NOT Conv_1_en_req THEN
						Feeder_Current_State	:= Wait_Pusher_Position;
					END_IF;

					IF F_Emergency_Stop THEN
						Feeder_Current_State 	:= Feeder_Stop_Seq;
					END_IF

					IF F_Immediate_Stop THEN
						En_Dis_Array[0] 		:= TRUE;
						Feeder_Old_State 		:= Feeder_Current_State;
						Feeder_Current_State 	:= Feeder_Stop_Seq;
					END_IF

				Wait_Pusher_Position:
					F_Current_State	:= 'Wait Pusher in Position';
					IF (I_IR_Sensor_1 OR (Sensor_Reached[0] AND Sensor_Memory[0])) THEN
						Sensor_Reached[0] 		:= FALSE;
						Sensor_Memory[0] 		:= FALSE;
						Conv_1_dis_req 			:= TRUE;
						Conv_2_en_req 			:= TRUE;
						Conv_3_en_req 			:= TRUE;
						Feeder_Current_State 	:= Layer_Check;
					END_IF

					IF F_Emergency_Stop THEN
						Feeder_Current_State 	:= Feeder_Stop_Seq;
					END_IF

					IF F_Immediate_Stop THEN
						Sensor_Memory[0] 		:= TRUE;
						En_Dis_Array[0] 		:= TRUE;
						Feeder_Old_State 		:= Feeder_Current_State;
						Feeder_Current_State 	:= Feeder_Stop_Seq;
					END_IF

				Layer_Check:
					F_Current_State	:= 'Layer Check';
					IF (NOT Conv_1_dis_req AND NOT Conv_2_en_req AND NOT Conv_3_en_req) THEN
						IF NOT C_Layer_Counter THEN
							IF Box_Counter < 8 THEN
								Turnpusher_dis_req 		:= TRUE;
								Pusher_en_req 			:= TRUE;
								Main_Line 				:= TRUE;
								Feeder_Current_State 	:= Line_Check;
							END_IF
							IF Box_Counter >= 8 THEN
								Turnpusher_en_req 		:= TRUE;
								Pusher_en_req 			:= TRUE;
								Main_Line 				:= FALSE;
								Feeder_Current_State 	:= Line_Check;
							END_IF
						END_IF

						IF C_Layer_Counter THEN
							IF Box_Counter < 6 THEN
								Turnpusher_en_req 		:= TRUE;
								Pusher_en_req 			:= TRUE;
								Main_Line 				:= FALSE;
								Feeder_Current_State 	:= Line_Check;
							END_IF
							IF Box_Counter >= 6 THEN
								Turnpusher_dis_req 		:= TRUE;
								Pusher_en_req 			:= TRUE;
								Main_Line 				:= TRUE;
								Feeder_Current_State 	:= Line_Check;
							END_IF
						END_IF
					END_IF

					IF F_Emergency_Stop THEN
						Feeder_Current_State 	:= Feeder_Stop_Seq;
					END_IF

					IF F_Immediate_Stop THEN
						En_Dis_Array[1] 		:= TRUE;
						En_Dis_Array[2] 		:= TRUE;
						En_Dis_Array[4] 		:= TRUE;
						Feeder_Old_State 		:= Feeder_Current_State;
						Feeder_Current_State 	:= Feeder_Stop_Seq;
					END_IF

				Line_Check:
					F_Current_State	:= 'Line Check';
					IF (NOT Turnpusher_dis_req AND NOT Pusher_en_req AND Main_Line) THEN
						Pusher_dis_req 			:= TRUE;
						Feeder_Current_State 	:= Wait_IR_Sensor_2;
					END_IF

					IF (NOT Turnpusher_en_req AND NOT Pusher_en_req AND NOT Main_Line) THEN
						Pusher_dis_req 			:= TRUE;
						Feeder_Current_State 	:= Wait_IR_Sensor_2;
					END_IF

					IF F_Emergency_Stop THEN
						Feeder_Current_State 	:= Feeder_Stop_Seq;
					END_IF

					IF F_Immediate_Stop THEN
						Sensor_Memory[1] 		:= TRUE;
						En_Dis_Array[2] 		:= TRUE;
						En_Dis_Array[4] 		:= TRUE;
						En_Dis_Array[6] 		:= TRUE;
						IF Main_Line THEN
							En_Dis_Array[9] 	:= TRUE;
						END_IF
						IF NOT Main_Line THEN
							En_Dis_Array[8] 	:= TRUE;
						END_IF
						Feeder_Old_State 		:= Feeder_Current_State;
						Feeder_Current_State 	:= Feeder_Stop_Seq;
					END_IF

				Wait_IR_Sensor_2:
					F_Current_State	:= 'Wait IR Sensor 2';
					IF ((I_IR_Sensor_2 OR (Sensor_Reached[1] AND Sensor_Memory[1])) AND NOT Pusher_dis_req) THEN
						Sensor_Reached[1] 		:= FALSE;
						Sensor_Memory[1] 		:= FALSE;
						Box_Counter 			:= Box_Counter + 1;
						Feeder_Current_State 	:= Box_In_Pos;
					END_IF

					IF F_Emergency_Stop THEN
						Feeder_Current_State 	:= Feeder_Stop_Seq;
					END_IF

					IF F_Immediate_Stop THEN
						Sensor_Memory[1] 		:= TRUE;
						En_Dis_Array[2] 		:= TRUE;
						En_Dis_Array[4] 		:= TRUE;
						En_Dis_Array[7] 		:= TRUE;
						Feeder_Old_State 		:= Feeder_Current_State;
						Feeder_Current_State 	:= Feeder_Stop_Seq;
					END_IF

				Box_In_Pos:
					F_Current_State	:= 'Box In Position';
					IF NOT C_Layer_Counter THEN
						IF (Box_Counter = 8 OR Box_Counter = 11 OR Box_Counter = 14) THEN
							Conv_2_dis_req 			:= TRUE;
							Feeder_Current_State 	:= Wait_Conveyor_Stop;
						ELSE
							Feeder_Current_State 	:= Wait_Start;
						END_IF
					END_IF

					IF C_Layer_Counter THEN
						IF (Box_Counter = 3 OR Box_Counter = 6 OR Box_Counter = 14) THEN
							Conv_2_dis_req 			:= TRUE;
							Feeder_Current_State 	:= Wait_Conveyor_Stop;
						ELSE
							Feeder_Current_State 	:= Wait_Start;
						END_IF
					END_IF

					IF F_Emergency_Stop THEN
						Feeder_Current_State 		:= Feeder_Stop_Seq;
					END_IF

					IF F_Immediate_Stop THEN
						En_Dis_Array[2] 		:= TRUE;
						En_Dis_Array[4] 		:= TRUE;
						Feeder_Old_State 		:= Feeder_Current_State;
						Feeder_Current_State 	:= Feeder_Stop_Seq;
					END_IF

				Wait_Conveyor_Stop:
					F_Current_State	:= 'Wait Conveyor Stop';
					IF NOT Conv_2_dis_req THEN
						IF Box_Counter = 14 THEN
							Feeder_Current_State 	:= Feeder_Idle;
						END_IF
						IF Box_Counter < 14 THEN
							End_Layer := FALSE;
							Carriage_Tar_Pos 		:= 0.44;
							Carriage.Axis_Command 	:= Change_Pos;
							Feeder_Current_State 	:= Carriage_FWD_Pos;
						END_IF
					END_IF

					IF F_Emergency_Stop THEN
						Feeder_Current_State 	:= Feeder_Stop_Seq;
					END_IF

					IF F_Immediate_Stop THEN
						En_Dis_Array[3] 		:= TRUE;
						En_Dis_Array[4] 		:= TRUE;
						Feeder_Old_State 		:= Feeder_Current_State;
						Feeder_Current_State 	:= Feeder_Stop_Seq;
					END_IF

				Feeder_Idle:
					F_Current_State	:= 'Feeder Idle';
					F_Ready 		:= TRUE;
					IF C_Layer_Counter THEN
						Second_Layer := TRUE;
					END_IF

					IF Load_Boxes_On_The_C THEN
						End_Layer 				:= TRUE;
						C_Layer_Counter 		:= NOT C_Layer_Counter;
						Carriage_Tar_Pos 		:= 1.1;
						Carriage.Axis_Command 	:= Change_Pos;
						Feeder_Current_State 	:= Carriage_FWD_Pos;
					END_IF

					IF F_Emergency_Stop THEN
						Feeder_Current_State 	:= Feeder_Stop_Seq;
					END_IF

					IF F_Immediate_Stop OR F_On_Phase_Stop THEN
						En_Dis_Array[4] 		:= TRUE;
						Feeder_Old_State 		:= Feeder_Current_State;
						Feeder_Current_State 	:= Feeder_Stop_Seq;
					END_IF

				Carriage_FWD_Pos:
					F_Current_State	:= 'Carriage In Forward Position';
					IF (Carriage_Pos_Reached OR Carriage_Pos_Restored) THEN
						Check_Pos 				:= FALSE;
						Carriage_Pos_Restored 	:= FALSE;
						Carriage.Axis_Command 	:= Idle;
						Feeder_Current_State 	:= Carriage_BWD_Pos;
					END_IF

					IF F_Emergency_Stop THEN
						Feeder_Current_State 	:= Feeder_Stop_Seq;
					END_IF

					IF F_Immediate_Stop THEN
						En_Dis_Array[4] 		:= TRUE;
						IF End_Layer THEN
							Check_Pos 	:= TRUE;
							Old_Pos 	:= 1.1;
						END_IF
						IF NOT End_Layer THEN
							Check_Pos 	:= TRUE;
							Old_Pos 	:= 0.44;
						END_IF
						Feeder_Old_State 		:= Feeder_Current_State;
						Feeder_Current_State 	:= Feeder_Stop_Seq;
					END_IF

				Carriage_BWD_Pos:
					F_Current_State	:= 'Carriage in Backward Position';
					IF NOT Carriage.Axis_In_Pos THEN
						Carriage_Tar_Pos 		:= 0.0;
						Carriage.Axis_Command 	:= Change_Pos;
						Feeder_Current_State 	:= Wait_Start_Pos;
					END_IF

					IF F_Emergency_Stop THEN
						Feeder_Current_State 	:= Feeder_Stop_Seq;
					END_IF

					IF F_Immediate_Stop THEN
						En_Dis_Array[4] 		:= TRUE;
						Feeder_Old_State 		:= Feeder_Current_State;
						Feeder_Current_State 	:= Feeder_Stop_Seq;
					END_IF

				Wait_Start_Pos:
					F_Current_State	:= 'Wait State Position';
					IF Box_Counter = 14 THEN
						Boxes_On_The_C 		:= TRUE;
						Box_Counter 		:= 0;
					END_IF

					IF (Carriage_Pos_Reached OR Carriage_Pos_Restored) THEN
						Check_Pos 				:= FALSE;
						Carriage_Pos_Restored 	:= FALSE;
						Carriage.Axis_Command 	:= Idle;
						Feeder_Current_State 	:= Wait_Start;
					END_IF

					IF F_Emergency_Stop THEN
						Feeder_Current_State 	:= Feeder_Stop_Seq;
					END_IF

					IF F_Immediate_Stop THEN
						En_Dis_Array[4] 		:= TRUE;
						Check_Pos 				:= TRUE;
						Old_Pos 				:= 0;
						Feeder_Old_State 		:= Feeder_Current_State;
						Feeder_Current_State 	:= Feeder_Stop_Seq;
					END_IF

			END_CASE

			IF I_IR_Sensor_1 THEN
				Sensor_Reached[0] := TRUE;
			END_IF

			IF I_IR_Sensor_2 THEN
				Sensor_Reached[1] := TRUE;
			END_IF

			//Conveyor_IF
			Conveyor_1(	Dev_Operation 		:= Operation_Type,
						Dev_Type 			:= Dev_Without_Feedback OR Dev_With_Single_Actuation,
						Dev_Clock 			:= TRUE,
						Dev_Enable_Time 	:= Conv_1_En_Time,
						Dev_Disable_Time	:= Conv_1_Dis_Time,
						Dev_Diagnose_Enable := TRUE,
						Dev_Enable_Preset 	:= FALSE,
						Dev_Enable_Request 	:= Conv_1_en_req,
						Dev_Disable_Request := Conv_1_dis_req);
			O_Conveyor_1		:= Conveyor_1.Dev_Enabled;
			e_Conveyor_1_Fault 	:= (*Conveyor_1.Dev_Actuator_Fault OR*) Conveyor_1_Fault_HMI;

			//Conveyor_Turn1
			Conveyor_2(	Dev_Operation 		:= Operation_Type,
						Dev_Type 			:= Dev_Without_Feedback OR Dev_With_Single_Actuation,
						Dev_Clock 			:= TRUE,
						Dev_Enable_Time 	:= Conv_2_En_Time,
						Dev_Disable_Time	:= Conv_2_Dis_Time,
						Dev_Diagnose_Enable := TRUE,
						Dev_Enable_Preset 	:= FALSE,
						Dev_Enable_Request 	:= Conv_2_en_req,
						Dev_Disable_Request := Conv_2_dis_req);
			O_Conveyor_2 		:= Conveyor_2.Dev_Enabled;
			e_Conveyor_2_Fault 	:= (*Conveyor_2.Dev_Actuator_Fault OR*) Conveyor_2_Fault_HMI;

			//Pusher
			Pusher_1(	Dev_Operation 		:= Operation_Type,
						Dev_Type 			:= Dev_With_Double_Feedback OR Dev_With_Single_Actuation,
						Dev_Enabled_Sensor 	:= I_Pusher_1_F,
						Dev_Disabled_Sensor := I_Pusher_1_B,
						Dev_Clock 			:= TRUE,
						Dev_Enable_Time 	:= Pusher_1_En_Time,
						Dev_Disable_Time	:= Pusher_1_Dis_Time,
						Dev_Diagnose_Enable := TRUE,
						Dev_Enable_Preset 	:= FALSE,
						Dev_Enable_Request 	:= Pusher_en_req,
						Dev_Disable_Request := Pusher_dis_req);
			O_Pusher_1 				:= Pusher_1.Dev_Enabled;
			e_Feeder_Pusher_Fault 	:= (*Pusher_1.Dev_Fault OR*) Pusher_1_Fault_HMI;

			//Conveoyr_end
			Conveyor_3(	Dev_Operation 		:= Operation_Type,
						Dev_Type 			:= Dev_Without_Feedback OR Dev_With_Single_Actuation,
						Dev_Clock 			:= TRUE,
						Dev_Enable_Time 	:= Conv_3_En_Time,
						Dev_Disable_Time	:= Conv_3_Dis_Time,
						Dev_Diagnose_Enable := TRUE,
						Dev_Enable_Preset 	:= FALSE,
						Dev_Enable_Request 	:= Conv_3_en_req,
						Dev_Disable_Request := Conv_3_dis_req);
			O_Conveyor_3 		:= Conveyor_3.Dev_Enabled;
			e_Conveyor_3_Fault 	:= (*Conveyor_3.Dev_Actuator_Fault OR*) Conveyor_3_Fault_HMI;

			//Turn_Pusher
			Turn_Pusher(	Dev_Operation 		:= Operation_Type,
							Dev_Type 			:= Dev_With_Double_Feedback OR Dev_With_Double_Actuation,
							Dev_Enabled_Sensor 	:= I_Turn_Push_B,
							Dev_Disabled_Sensor := I_Turn_Push_F,
							Dev_Clock 			:= TRUE,
							Dev_Enable_Time 	:= Turn_Pusher_En_Time,
							Dev_Disable_Time	:= Turn_Pusher_Dis_Time,
							Dev_Diagnose_Enable := TRUE,
							Dev_Enable_Preset 	:= FALSE,
							Dev_Enable_Request 	:= Turnpusher_en_req,
							Dev_Disable_Request := Turnpusher_dis_req);
			O_Turn_Pusher_OFF		:= Turn_Pusher.Dev_Enabled;
			O_Turn_Pusher_ON		:= Turn_Pusher.Dev_Disabled;
			e_Turn_Pusher_Fault 	:= (*Turn_Pusher.Dev_Fault OR*) Turn_Pusher_Fault_HMI;

			//Carriage
			Carriage(	Axis_Act_Position 	:= I_Carriage_Push_Act_Pos,
						New_Set_Point 		:= Carriage_Tar_Pos,
						Axis_Dev_Timer 		:= 400,
						Axis_TGT_Sensor 	:= I_Carriage_Push_Tar_Rec);
			O_Carriage_Tar_Pos 		:= Carriage.Axis_TGT_Position;
			Carriage_Pos_Reached 	:= Carriage.Axis_In_Pos;
			e_Carriage_Fault 		:= (*Carriage.Axis_Dev_Fault OR*) Carriage_Fault_HMI;

		1: //Service Mode
			//Actuation Servicing
			IF NOT Service_Mode THEN
				State := 0;
			END_IF

			O_Conveyor_1 		:= Conveyor_1_HMI;
			IF NOT O_Conveyor_1 THEN
				O_Conveyor_1 	:= Conveyor_1_Jog_HMI;
			END_IF
			O_Conveyor_2 		:= Conveyor_2_HMI;
			IF NOT O_Conveyor_2 THEN
				O_Conveyor_2 	:= Conveyor_2_Jog_HMI;
			END_IF
			O_Conveyor_3 		:= Conveyor_3_HMI;
			IF NOT O_Conveyor_3 THEN
				O_Conveyor_3 	:= Conveyor_3_Jog_HMI;
			END_IF
			O_Pusher_1 		:= Pusher_1_HMI;
			IF NOT O_Pusher_1 THEN
				O_Pusher_1 	:= Pusher_1_Jog_HMI;
			END_IF

			O_Turn_Pusher_ON 	:= Turn_Pusher_ON_HMI;
			O_Turn_Pusher_OFF 	:= Turn_Pusher_OFF_HMI;

			Carriage_Tar_Pos_Dis_HMI 	:= Carriage_Target_Pos_HMI;
			IF Carriage_Push_Origin_HMI THEN
				O_Carriage_Tar_Pos 		:= 0.0;
			ELSIF Carriage_Push_Target_HMI THEN
				O_Carriage_Tar_Pos 		:= Carriage_Target_Pos_HMI;
			END_IF

			//Sensor Servicing
			IR1_HMI 						:= I_IR_Sensor_1;
			IR2_HMI 						:= I_IR_Sensor_2;
			Turn_Pusher_F_HMI 				:= I_Turn_Push_B;
			Turn_Pusher_B_HMI 				:= I_Turn_Push_F;
			Pusher_1_F_HMI 					:= I_Pusher_1_F;
			Pusher_1_B_HMI 					:= I_Pusher_1_B;
			Carriage_Push_TarRech_HMI 		:= I_Carriage_Push_Tar_Rec;
			Carriage_Push_ActPos_Dis_HMI 	:= I_Carriage_Push_Act_Pos;

	END_CASE

END_PROGRAM

PROGRAM _EXIT
	(* Insert code here *)

END_PROGRAM
```

### Program Logical/Crane (IEC)

#### Types.typ
```iecst
TYPE
	Crane_State :
		(
		Crane_Stop_Seq := 1,
		Crane_Stop_Done := 2,
		Reset_Crane_Config := 3,
		Restore_Crane_Config_1 := 4,
		Restore_Crane_Config_2 := 5,
		Restore_Crane_Config_3 := 6,
		Wait_Start := 7,
		Wait_Gantry_Crane_Start_Pos := 8,
		Wait_Cartboard_Load_Pos := 9,
		Wait_Cartboard_Load := 10,
		Wait_Box_Crane_Start_Pos := 11,
		Wait_Pusher_Z_Start_Pos_Down := 12,
		Wait_Pusher_X_Start_Pos_FWD := 13,
		Lock_Cartboard := 14,
		Wait_Boxes := 15,
		Wait_SlideRail_Hold := 16,
		Wait_Pusher_Z_Push_Pos_Up := 17,
		Wait_Pusher_X_Push_Pos_BKW := 18,
		Crane_Idle := 19,
		Wait_Pusher_Z_Push_Pos_Down := 20,
		Wait_Box_Crane_Cartboard_Pos := 21,
		Wait_Gantry_Crane_Cartboard_Pos := 22,
		Place_Cartboard := 23,
		Place_Boxes := 24,
		Open_SlideRail := 25,
		Pusher_FWD := 26
		);
END_TYPE
```

#### Variables.var
```iecst
VAR
	State : USINT := 0;
	Crane_Current_State : Crane_State;
END_VAR
(*Gantry Crane*)
VAR
	Gantry_Crane : Gen_Axis;
	Gantry_Crane_Pos_Reached : BOOL;
	Gantry_Crane_Tar_Pos : REAL;
END_VAR
(*Box Crane*)
VAR
	Box_Crane : Gen_Axis;
	Box_Crane_Pos_Reached : BOOL;
	Box_Crane_Tar_Pos : REAL;
END_VAR
(*Cartboard*)
VAR
	Cartboard : Gen_Device;
	Cartboard_En_Time : INT := 60;
	Cartboard_Dis_Time : INT := 60;
END_VAR
(*Vacuum*)
VAR
	Vacuum : Gen_Device;
	Vacuum_En_Time : INT := 80;
	Vacuum_Dis_Time : INT := 80;
END_VAR
(*SlideRail*)
VAR
	Box_Holder : Gen_Device;
	Box_Holder_En_Time : INT := 60;
	Box_Holder_Dis_Time : INT := 60;
END_VAR
(*Pusher X*)
VAR
	Pusher_X : Gen_Device;
	Pusher_X_En_Time : INT := 60;
	Pusher_X_Dis_Time : INT := 60;
END_VAR
(*Pusher Z*)
VAR
	Pusher_Z : Gen_Device;
	Pusher_Z_En_Time : INT;
	Pusher_Z_Dis_Time : INT;
END_VAR
(*Faults*)
VAR
	En_Dis_Array : ARRAY[0..9] OF BOOL := [10(FALSE)];
	a : INT := 0;
	En_Dis_Counter : INT;
	Check_Pos : ARRAY[0..1] OF BOOL := [2(FALSE)];
	Old_Pos : ARRAY[0..1] OF REAL;
	Box_Crane_Pos_Restored : BOOL := FALSE;
	Gantry_Crane_Pos_Restored : BOOL := FALSE;
	Old_State : Crane_State;
	Stop_Req : BOOL := FALSE;
END_VAR
VAR CONSTANT
	Idle : WORD := 0;
	Change_Vel : WORD := 1;
	Change_Pos : WORD := 2;
	Emergency_Stop_Req : WORD := 3;
END_VAR
VAR
	Vacuum_En_Req : BOOL;
	Vacuum_Dis_Req : BOOL;
	Cartboard_En_Req : BOOL;
	Cartboard_Dis_Req : BOOL;
	Box_Holder_En_Req : BOOL;
	Box_Holder_Dis_Req : BOOL;
	Pusher_Z_En_Req : BOOL;
	Pusher_Z_Dis_Req : BOOL;
	Pusher_X_En_Req : BOOL;
	Pusher_X_Dis_Req : BOOL;
	New_Variable2 : USINT;
	New_Variable1 : USINT;
	New_Variable : USINT;
END_VAR
```
